(* Logix 5000 project; controller Sucrose_Main Emulate 5570 rev 20.12; software revision 20.01; part 3 of 30 *)
(* tags used below, declared in another part *)
   CIPRemote : Area_Program;
   DATE_TIME : Date_Time;
   Rung_Comment : BOOL;
   SucroseCIP_FILTRATION_ALL_PATHS_Selected : BOOL;
   SucroseCIP_FILTRATION_PATH1_Selected : BOOL;
   SucroseCIP_FILTRATION_PATH2_Selected : BOOL;
   SucroseCIP_FILTRATION_PATH3_Selected : BOOL;
   SucroseCIP_FILTRATION_PATH4_Selected : BOOL;
   SucroseCIP_FILTRATION_REMOTE : CIP_REMOTE;
   SucroseCIP_P230401_REMOTE : CIP_REMOTE;
   SucroseCIP_P230402_REMOTE : CIP_REMOTE;
   SucroseCIP_PAUSED : BOOL;
   SucroseCIP_RECEIVING2_REMOTE : CIP_REMOTE;
   SucroseCIP_RINGMAIN_REMOTE : CIP_REMOTE;
   SucroseCIP_RUNNING : BOOL;
   SucroseCIP_SeatLift_Pulsing : BOOL;
   SucroseFiltration : Area_Program;

        .TMR_LOGIC[5]   // AIR BLOW TIMER
        .CALC_LOGIC[0]   // PRE-FILTER 1 DIFF PRESSURE
        .CALC_LOGIC[1]   // PRE-FILTER 2 DIFF PRESSURE
        .BIT_LOGIC[2].2   // FINAL FILTER 1 SIP STARTED
        .BIT_LOGIC[2].3   // FINAL FILTER 2 SIP STARTED
        .BIT_LOGIC[1].4   // BACKFLUSH ROUTINE ACTIVE
        .BIT_LOGIC[1].5   // AIR BLOW STEP 1 ACTIVE
        .BIT_LOGIC[1].6   // AIR BLOW STEP 2 ACTIVE
        .BIT_LOGIC[1].7   // AIR BLOW STEP 3 ACTIVE
        .BIT_LOGIC[1].8   // INITIAL AIR BLOW COMPLETE
        .BIT_LOGIC[2].0   // PRE FILTER 1 SIP STARTED
        .BIT_LOGIC[0].10   // OK TO START TRANSFER PUMP
        .BIT_LOGIC[1].10   // OK TO START BACKFLUSH PUMP
        .BIT_LOGIC[2].1   // PRE FILTER 2 SIP STARTED
        .BIT_LOGIC[2].5   // SIP STEP ACTIVE
        .BIT_LOGIC[0].5   // PRE FILTER 1 FINAL FILTER 1 PATH ENABLED FOR PRODUCTION
        .BIT_LOGIC[1].17   // AIR BLOW ACTIVE
        .BIT_LOGIC[2].6   // SIP STEP COMPLETE
        .BIT_LOGIC[0].6   // PRE FILTER 1 FINAL FILTER 2 PATH ENABLED FOR PRODUCTION
        .BIT_ALARM[0].11   // FINAL FILTER 1 DIFF PRESSURE ABOVE 40 ALARM
        .BIT_ALARM[0].15   // FINAL FILTER 2 DIFF PRESSURE ABOVE 40 ALARM
        .TMR_ALARM[0]   // PRE FILTER 1 DIFF PRESSURE ABOVE 16 ALARM TIMER
        .BIT_LOGIC[1].0   // PRE FILTER 1 BACKFLUSH STARTED
        .BIT_ALARM[0].0   // PRE FILTER 1 DIFF PRESSURE ABOVE 16 ALARM
        .BIT_ALARM[0].1   // PRE FILTER 1 DIFF PRESSURE ABOVE 20 ALARM
        .BIT_ALARM[0].2   // PRE FILTER 1 DIFF PRESSURE ABOVE 6 ALARM
        .TMR_ALARM[2]   // PRE FILTER 1 DIFF PRESSURE ABOVE 6 ALARM TIMER
        .TMR_ALARM[3]   // PRE FILTER 1 DIFF PRESSURE ABOVE 40 ALARM TIMER
        .BIT_ALARM[0].3   // PRE FILTER 1 DIFF PRESSURE ABOVE 40 ALARM
        .BIT_LOGIC[0].7   // PRE FILTER 2 FINAL FILTER 1 PATH ENABLED FOR PRODUCTION
        .BIT_LOGIC[0].8   // PRE FILTER 2 FINAL FILTER 2 PATH ENABLED FOR PRODUCTION
        .TMR_ALARM[4]   // PRE FILTER 2 DIFF PRESSURE ABOVE 16 ALARM
        .BIT_LOGIC[1].1   // PRE FILTER 2 BACKFLUSH STARTED
        .TMR_ALARM[5]   // PRE FILTER 2 DIFF PRESSURE ABOVE 20 ALARM
        .TMR_ALARM[6]   // PRE FILTER 2 DIFF PRESSURE ABOVE 6 ALARM
        .TMR_ALARM[7]   // PRE FILTER 2 DIFF PRESSURE ABOVE 40 ALARM
        .CALC_LOGIC[2]   // FINAL FILTER 1 DIFF PRESSURE
        .TMR_ALARM[8]   // FINAL FILTER 1 DIFF PRESSURE ABOVE 16 ALARM
        .BIT_LOGIC[1].2   // FINAL FILTER 1 BACKFLUSH STARTED
        .TMR_ALARM[10]   // FINAL FILTER 1 DIFF PRESSURE ABOVE 6 ALARM
        .TMR_ALARM[11]   // FINAL FILTER 1 DIFF PRESSURE ABOVE 40 ALARM
        .CALC_LOGIC[3]   // FINAL FILTER 2 DIFF PRESSURE
        .TMR_ALARM[12]   // FINAL FILTER 2 DIFF PRESSURE ABOVE 16 ALARM
        .BIT_LOGIC[1].3   // FINAL FILTER 2 BACKFLUSH STARTED
        .TMR_ALARM[14]   // FINAL FILTER 2 DIFF PRESSURE ABOVE 6 ALARM
        .BIT_ALARM[0].7   // PRE FILTER 2 DIFF PRESSURE ABOVE 40 ALARM
        .TMR_ALARM[1]   // PRE FILTER 1 DIFF PRESSURE ABOVE 20 ALARM TIMER
        .TMR_ALARM[9]   // FINAL FILTER 1 DIFF PRESSURE ABOVE 20 ALARM
        .TMR_ALARM[13]   // FINAL FILTER 2 DIFF PRESSURE ABOVE 20 ALARM
        .TMR_ALARM[15]   // FINAL FILTER 2 DIFF PRESSURE ABOVE 40 ALARM
        .BIT_LOGIC[0].0   // FILTRATION SKID IN PRODUCTION MODE
        .BIT_LOGIC[0].1   // PRE-FILTER 1 READY FOR PRODUCTION
        .BIT_LOGIC[0].2   // PRE-FILTER 2 READY FOR PRODUCTION
        .BIT_LOGIC[0].3   // FINAL FILTER 1 READY FOR PRODUCTION
        .BIT_LOGIC[0].4   // FINAL FILTER 2 READY FOR PRODUCTION
        .BIT_LOGIC[0].9   // OPEN VENT VALVES ON SELECTED FILTERS
        .BIT_LOGIC[1].9   // BACKFLUSH ROUTINE HOT FLUSH STEP ACTIVE
        .BIT_LOGIC[1].11   // SEND FLUSH TO SCRAP
        .BIT_LOGIC[1].12   // BACKFLUSH DRAIN STEP ACTIVE
        .BIT_LOGIC[1].13   // PRE FILTER 1 CIP BACKFLUSH COMPLETE INTERLOCK TO CIP SKID
        .BIT_LOGIC[1].14   // PRE FILTER 2 CIP BACKFLUSH COMPLETE INTERLOCK TO CIP SKID
        .BIT_LOGIC[1].15   // FINAL FILTER 1 CIP BACKFLUSH COMPLETE INTERLOCK TO CIP SKID
        .BIT_LOGIC[1].16   // FINAL FILTER 2 CIP BACKFLUSH COMPLETE INTERLOCK TO CIP SKID
        .BIT_LOGIC[1].18   // FILTER BACKFLUSH FOR CIP SELECTED
        .BIT_LOGIC[2].4   // STAND ALONE SIP SEQUENCE SELECTED
        .BIT_LOGIC[3].0   // AIR INTEGRITY TEST STARTED FOR FINAL FILTER 1
        .BIT_LOGIC[3].1   // AIR INTEGRITY TEST STARTED FOR FINAL FILTER 2
        .BIT_LOGIC[3].2   // FINAL FILTER INTEGRITY TEST ACTIVE
        .BIT_LOGIC[3].3   // FINAL FILTER INTEGRITY TEST FAILED
        .BIT_LOGIC[3].4   // FINAL FILTER INTEGRITY TEST COMPLETE
        .BIT_LOGIC[3].5   // FINAL FILTER 1 INTEGRITY TEST SELECTED
        .BIT_LOGIC[3].6   // FINAL FILTER 2 INTEGRITY TEST SELECTED
        .TMR_LOGIC[0]   // INITIAL FILTRATION VENTING TIMER
        .TMR_LOGIC[1]   // VENTING AFTER TRANSFER PUMP TIMER
        .TMR_LOGIC[6]   // BACKFLUSH INITIAL FILTRATION VENTING TIMER
        .TMR_LOGIC[7]   // DELAY TO CLOSE VENT VALVE TIMER
        .TMR_LOGIC[8]   // BACKFLUSH SEQUENCE FLUSH ACTIVE TIMER
        .TMR_LOGIC[9]   // BACKFLUSH DRAIN SYSTEM TIMER
        .TMR_LOGIC[10]   // SIP SEQUENCE 250 DEG TIMER
        .TMR_LOGIC[11]   // INITIAL AIR INTEGRITY TEST TIMER
        .TMR_LOGIC[12]   // AIR INTEGRITY TEST ACTIVE TIMER
        .TMR_LOGIC[13]   // SIP SEQUENCE 254 DEG TIMER
        .TMR_LOGIC[14]   // SIP SEQUENCE BELOW TEMP TIMER
        .TMR_LOGIC[15]   // DELAY AFTER CLOSING STEAM VALVE
        .CTR_LOGIC[0]   // PRE FILTER 1 BACKFLUSH COUNTER
        .CTR_LOGIC[1]   // PRE FILTER 2 BACKFLUSH COUNTER
        .CTR_LOGIC[2]   // FINAL FILTER 1 BACKFLUSH COUNTER
        .CTR_LOGIC[3]   // FINAL FILTER 2 BACKFLUSH COUNTER
        .BIT_HMI[0].0   // PRE-FILTER 1 WITH FINAL FILTER 1PATH SELECTED PB
        .BIT_HMI[0].1   // PRE-FILTER 1 WITH FINAL FILTER 2 PATH SELECTED PB
        .BIT_HMI[0].2   // PRE-FILTER 2 WITH FINAL FILTER 1PATH SELECTED PB
        .BIT_HMI[0].3   // PRE-FILTER 2 WITH FINAL FILTER 2 PATH SELECTED PB
        .BIT_HMI[0].4   // FILTER INSTALLED IN PRE FILTER 1 HMI CONFIRMATION
        .BIT_HMI[0].5   // FILTER INSTALLED IN PRE FILTER 2 HMI CONFIRMATION
        .BIT_HMI[0].6   // FILTER INSTALLED IN FINAL FILTER 1 HMI CONFIRMATION
        .BIT_HMI[0].7   // FILTER INSTALLED IN FINAL FILTER 2 HMI CONFIRMATION
        .BIT_HMI[0].8   // PRE FILTER 1 YELLOW FLASHING WARNING ON HMI
        .BIT_HMI[0].9   // PRE FILTER 2 YELLOW FLASHING WARNING ON HMI
        .BIT_HMI[0].10   // FINAL FILTER 1 YELLOW FLASHING WARNING ON HMI
        .BIT_HMI[0].11   // FINAL FILTER 2 YELLOW FLASHING WARNING ON HMI
        .BIT_HMI[0].12   // PRE FILTER 1 RED FLASHING ALARM ON HMI
        .BIT_HMI[0].13   // PRE FILTER 2 RED FLASHING ALARM ON HMI
        .BIT_HMI[0].14   // FIANL FILTER 1 RED FLASHING ALARM ON HMI
        .BIT_HMI[0].15   // FIANL FILTER 2 RED FLASHING ALARM ON HMI
        .BIT_HMI[0].16   // PROMPT FOR PRE FILTER 1 FILTER INSTALLED VISIBILITY
        .BIT_HMI[0].17   // PROMPT FOR PRE FILTER 2 FILTER INSTALLED VISIBILITY
        .BIT_HMI[0].18   // PROMPT FOR FINAL FILTER 1 FILTER INSTALLED VISIBILITY
        .BIT_HMI[0].19   // PROMPT FOR FINAL FILTER 2 FILTER INSTALLED VISIBILITY
        .BIT_HMI[0].20   // PROMPT FOR PRE FILTER 1 FILTER NOT INSTALLED VISIBILITY
        .BIT_HMI[0].21   // PROMPT FOR PRE FILTER 2 FILTER NOT INSTALLED VISIBILITY
        .BIT_HMI[0].22   // PROMPT FOR FINAL FILTER 1 FILTER NOT INSTALLED VISIBILITY
        .BIT_HMI[0].23   // PROMPT FOR FINAL FILTER 2 FILTER NOT INSTALLED VISIBILITY
        .BIT_HMI[0].24   // FILTER SEQUENCE STARTED DISABLE FILTER SELECTION VISABILITY
        .BIT_HMI[0].25   // PROMPT FOR PRE FILTER 1 NEW FILTER INSTALLED VISIBILITY
        .BIT_HMI[0].26   // PROMPT FOR PRE FILTER 2 NEW FILTER INSTALLED VISIBILITY
        .BIT_HMI[0].27   // PROMPT FOR FINAL FILTER 1 NEW FILTER INSTALLED VISIBILITY
        .BIT_HMI[0].28   // PROMPT FOR FINAL FILTER 2 NEW FILTER INSTALLED VISIBILITY
        .BIT_HMI[1].0   // FILTER ROUTINE START PB
        .BIT_HMI[1].1   // BACKFLUSH ROUTINE ABORT PB
        .BIT_HMI[1].2   // FILTER ROUTINE PAUSE PB
        .BIT_HMI[1].5   // PRE FILTER 1 SELECTED FOR BACKFLUSH
        .BIT_HMI[1].6   // PRE FILTER 2 SELECTED FOR BACKFLUSH
        .BIT_HMI[1].7   // FINAL FILTER 1 SELECTED FOR BACKFLUSH
        .BIT_HMI[1].8   // FINAL FILTER 2 SELECTED FOR BACKFLUSH
        .BIT_HMI[1].10   // PRE FILTER 1 SELECTED FOR CIP BACKFLUSH
        .BIT_HMI[1].11   // PRE FILTER 2 SELECTED FOR CIP BACKFLUSH
        .BIT_HMI[1].12   // FINAL FILTER 1 SELECTED FOR CIP BACKFLUSH
        .BIT_HMI[1].13   // FINAL FILTER 2 SELECTED FOR CIP BACKFLUSH
        .BIT_HMI[2].0   // SIP ROUTINE START PB
        .BIT_HMI[2].1   // SIP ROUTINE ABORT PB
        .BIT_HMI[2].5   // PRE FILTER 1 SELECTED FOR SIP
        .BIT_HMI[2].6   // PRE FILTER 2 SELECTED FOR SIP
        .BIT_HMI[2].7   // FINAL FILTER 1 SELECTED FOR SIP
        .BIT_HMI[2].8   // FINAL FILTER 2 SELECTED FOR SIP
        .BIT_HMI[3].0   // AIR INTEGRITY TEST START PB
        .BIT_HMI[3].1   // AIR INTEGRITY TEST ABORT PB
        .BIT_HMI[3].5   // FINAL FILTER 1 SELECTED FOR AIR INTEGRITY TEST
        .BIT_HMI[3].6   // FINAL FILTER 2 SELECTED FOR AIR INTEGRITY TEST
        .STATUS_HMI[1]   // PREFILTER 1 STATUS 0=PROD, 1=AIRBLOW, 2=BACKFLUSH, 3=SIP, 4=INTERG TEST, 5=CIP, 6=SERVICE
        .STATUS_HMI[2]   // PREFILTER 2 STATUS 0=PROD, 1=AIRBLOW, 2=BACKFLUSH, 3=SIP, 4=INTERG TEST, 5=CIP, 6=SERVICE
        .STATUS_HMI[3]   // FINAL FILTER 1 STATUS 0=PROD, 1=AIRBLOW, 2=BACKFLUSH, 3=SIP, 4=INTERG TEST, 5=CIP, 6=SERVICE
        .STATUS_HMI[4]   // FINAL FILTER 2 STATUS 0=PROD, 1=AIRBLOW, 2=BACKFLUSH, 3=SIP, 4=INTERG TEST, 5=CIP, 6=SERVICE
   SucroseReceiving : Area_Program := (TMR_Alarm[0].PRE := 15000, TMR_Alarm[1].PRE := 15000, TMR_Logic[3].PRE := 3000, TMR_Logic[4].PRE := 5000, TMR_Logic[5].PRE := 45000);
        .BIT_LOGIC[0].0   // SUCROSE TANKER QC APPROVED FOR RECEIVING
        .BIT_LOGIC[0].12   // PIG RETURN SEQUENCE ACTIVE
        .BIT_HMI[0].1   // SUCROSE TANKER START TRANSFER PUSHBUTTON PRESSED
        .BIT_HMI[0].2   // STOP TRANSFER REQUEST TO TANKER PUSHBUTTON PRESSED
        .BIT_LOGIC[0].2   // SUCROSE SUPPLY WATER PURGE ENABLED
        .BIT_LOGIC[0].4   // SUCROSE SUPPLY RECEIVING LINE FLUSH COMPLETE BIT
        .BIT_LOGIC[0].5   // SUCROSE SUPPLY RECEIVING LINE WATER PURGE COMPLETE
        .BIT_LOGIC[0].6   // SUCROSE SUPPLY RECEIVING LINE WATER PURGE PREVENT TANK VALVE FROM OPENING
        .BIT_LOGIC[0].7   // PIG LAUNCH SEQUENCE ACTIVE
        .BIT_LOGIC[0].8   // PLACE PIG IN LAUNCH POSITION
        .BIT_LOGIC[0].9   // ACTIVATE V3.1 VALVE TO SET PIG IN POSITION
        .BIT_LOGIC[0].10   // LAUNCH PIG BIT
        .BIT_LOGIC[0].11   // PIG AT RECEIVING STATION
        .BIT_LOGIC[0].13   // PIG BACK IN LAUNCHER. MOVE INTO PRODUCTION POSITION
        .BIT_LOGIC[0].14   // PIG IN PRODUCTION/CIP POSITION BIT
        .TMR_LOGIC[0]   // SUCROSE SUPPLY FLUSH TOTALIZER TIMER
        .TMR_LOGIC[1]   // SUCROSE SUPPLY WATER PURGE TOTALIZER TIMER
        .TMR_LOGIC[2]   // SUCROSE SUPPLY WATER PURGE DELAY SHUTOFF TIMER
        .TMR_LOGIC[3]   // DELAY TO ACTIVATE V3.1 VALVE
        .TMR_LOGIC[4]   // DELAY TO RETURN PIG TO LAUNCHER
        .TMR_LOGIC[5]   // PIPE VENTING TIMER
        .BIT_HMI[0].0   // SUCROSE TANKER QC APPROVED FOR RECEIVING PUSHBUTTON PRESSED
        .BIT_HMI[0].3   // HMI SUCROSE SUPPLY WATER PURGE PUSHBUTTON
        .BIT_HMI[0].4   // LAUNCH PIG HMI PB
        .BIT_HMI[0].5   // START SUCROSE RECEIVING PUMP HMI PB
        .BIT_HMI[1].1   // HMI SUCROSE TANK 1 DISCHARGE ENABLED PUSHBUTTON PRESSED
        .BIT_LOGIC[1].0   // TANK 1 RECEIVING FOR PIG LAUNCH
        .BIT_LOGIC[2].0   // TANK 2 RECEIVING FOR PIG LAUNCH
        .BIT_LOGIC[3].0   // TANK 3 RECEIVING FOR PIG LAUNCH
        .BIT_ALARM[0].0   // RECEIVING LINE NO FLOW, STOP PUMP 1
        .BIT_LOGIC[0].1   // ENABLE SUCROSE RECEIVING PUMP 1
        .BIT_HMI[0].9   // START SUCROSE RECEIVING PUMP 2 HMI PB
        .BIT_LOGIC[0].3   // ENABLE SUCROSE RECEIVING PUMP 2
        .BIT_HMI[0].10   // STOP SUCROSE RECEIVING PUMP 2 HMI PB
        .BIT_HMI[0].8   // USE PLANT PUMP 1 TO RECEIVE SUCROSE SELECTED PB
        .BIT_HMI[0].6   // STOP SUCROSE RECEIVING PUMP 1 HMI PB
        .BIT_HMI[0].11   // USE PLANT PUMP 2 TO RECEIVE SUCROSE SELECTED PB
        .BIT_ALARM[0].1   // RECEIVING LINE NO FLOW, STOP PUMP 2
   SucroseReturn : Area_Program;
   SucroseTanks : Area_Program := (TMR_Alarm[0].PRE := 6000, TMR_Alarm[1].PRE := 3000, TMR_Alarm[2].PRE := 3000, TMR_Alarm[3].PRE := 3000, TMR_Alarm[4].PRE := 30000, TMR_Alarm[5].PRE := 30000, TMR_Alarm[6].PRE := 30000, TMR_Alarm[7].PRE := 30000, TMR_Alarm[8].PRE := 30000, TMR_Alarm[9].PRE := 30000, TMR_Alarm[19].PRE := 5000, TMR_Alarm[20].PRE := 5000, TMR_Alarm[21].PRE := 5000, TMR_Alarm[22].PRE := 5000, TMR_Alarm[23].PRE := 5000, TMR_Alarm[24].PRE := 5000, TMR_Logic[0].PRE := 20000, TMR_Logic[1].PRE := 40000, TMR_Logic[2].PRE := 40000, TMR_Logic[3].PRE := 40000, TMR_Logic[9].PRE := 900000, TMR_Logic[10].PRE := 900000, TMR_Logic[11].PRE := 15000);
        .BIT_LOGIC[3].0   // SUCROSE TANK 3 OK TO RECEIVE TANKER
        .BIT_HMI[2].0   // HMI SUCROSE TANK 2 SELECTED TO RECEIVE TANKER PUSHBUTTON PRESSED
        .BIT_ALARM[0].10   // HTR_76_01_01 HIGH TEMPERATURE ALARM LATCH
        .BIT_LOGIC[1].3   // SUCROSE TANK 1 DISCHARGE ENABLED
        .BIT_LOGIC[1].9   // SUCROSE TANK 1 HEALOUT ENABLED
        .BIT_HMI[3].0   // HMI SUCROSE TANK 3 SELECTED TO RECEIVE TANKER PUSHBUTTON PRESSED
        .BIT_LOGIC[3].1   // SUCROSE TANK 3 TANK IN USE RECEIVING TANKER
        .BIT_LOGIC[1].12   // TANK
        .BIT_LOGIC[3].5   // SUCROSE TANK 3 DISCHARGE ACTIVE
        .BIT_ALARM[0].14   // HTR_76_02_01 LOW TEMPERATURE ALARM LATCH
        .BIT_LOGIC[1].1   // SUCROSE TANK 1 TANK IN USE RECEIVING TANKER
        .BIT_ALARM[0].13   // HTR_76_01_01 LOW TEMPERATURE ALARM LATCH
        .BIT_HMI[1].0   // HMI SUCROSE TANK 1 SELECTED TO RECEIVE TANKER PUSHBUTTON PRESSED
        .BIT_ALARM[0].16   // HTR_76_01_01 LOW FLOW ALARM LATCH
        .BIT_LOGIC[2].2   // SUCROSE TANK 2 READY TO RECEIVE TANKER
        .BIT_LOGIC[1].2   // SUCROSE TANK 1 READY TO RECEIVE TANKER
        .BIT_LOGIC[2].0   // SUCROSE TANK 2 OK TO RECEIVE TANKER
        .BIT_LOGIC[1].5   // SUCROSE TANK 1 DISCHARGE ACTIVE
        .BIT_ALARM[1].3   // TK_23_01_01 SELECTED TANK TOO FULL TO RECEIVE ALARM LATCH
        .BIT_LOGIC[1].0   // SUCROSE TANK 1 OK TO RECEIVE TANKER
        .BIT_LOGIC[3].2   // SUCROSE TANK 3 READY TO RECEIVE TANKER
        .BIT_LOGIC[2].5   // SUCROSE TANK 2 DISCHARGE ACTIVE
        .BIT_LOGIC[2].1   // SUCROSE TANK 2 TANK IN USE RECEIVING TANKER
        .BIT_ALARM[0].11   // HTR_76_02_01 HIGH TEMPERATURE ALARM LATCH
        .BIT_LOGIC[1].4   // TK_23_01_01 READY TO DISCHARGE
        .BIT_ALARM[0].17   // HTR_76_02_01 LOW FLOW ALARM LATCH
        .BIT_ALARM[1].13   // TK_23_02_01 SELECTED TANK TOO FULL TO RECEIVE ALARM LATCH
        .BIT_ALARM[0].12   // HTR_76_03_01 HIGH TEMPERATURE ALARM LATCH
        .BIT_ALARM[0].15   // HTR_76_03_01 LOW TEMPERATURE ALARM LATCH
        .BIT_ALARM[0].18   // HTR_76_03_01 LOW FLOW ALARM LATCH
        .BIT_HMI[1].1   // HMI SUCROSE TANK 1 DISCHARGE ENABLED PUSHBUTTON PRESSED
        .BIT_HMI[2].1   // HMI SUCROSE TANK 2 DISCHARGE ENABLED PUSHBUTTON PRESSED
        .BIT_LOGIC[2].3   // SUCROSE TANK 2 DISCHARGE ENABLED
        .BIT_HMI[3].1   // HMI SUCROSE TANK 3 DISCHARGE ENABLED PUSHBUTTON PRESSED
        .BIT_LOGIC[3].3   // SUCROSE TANK 3 DISCHARGE ENABLED
        .BIT_HMI[1].5   // HMI SUCRSOE TANK 1 HEALOUT ENABLED BIT
        .BIT_LOGIC[2].9   // SUCROSE TANK 2 HEALOUT ENABLED
        .BIT_LOGIC[3].9   // SUCROSE TANK 3 HEALOUT ENABLED
        .BIT_HMI[2].5   // HMI SUCRSOE TANK 2 HEALOUT ENABLED BIT
        .BIT_HMI[3].5   // HMI SUCRSOE TANK 3 HEALOUT ENABLED BIT
        .BIT_LOGIC[2].4   // TK_23_02_01 READY TO DISCHARGE
        .BIT_LOGIC[3].4   // TK_23_03_01 READY TO DISCHARGE
        .BIT_HMI[1].2   // HMI TK_23_01_01 PRIME TO P_23_01_01 PUSHBUTTON PRESSED
        .BIT_LOGIC[2].6   // TK_23_02_01 PRIME ENABLED FOR P_23_01_01 PATH
        .BIT_LOGIC[3].6   // TK_23_03_01 PRIME ENABLED FOR P_23_01_01 PATH
        .BIT_LOGIC[1].6   // TK_23_01_01 PRIME ENABLED FOR P_23_01_01 PATH
        .BIT_HMI[1].3   // HMI TK_23_01_01 PRIME TO P_23_01_02 PUSHBUTTON PRESSED
        .BIT_LOGIC[2].7   // TK_23_02_01 PRIME ENABLED FOR P_23_01_02 PATH
        .BIT_LOGIC[3].7   // TK_23_03_01 PRIME ENABLED FOR P_23_01_02 PATH
        .BIT_LOGIC[1].7   // TK_23_01_01 PRIME ENABLED FOR P_23_01_02 PATH
        .BIT_HMI[2].2   // HMI TK_23_02_01 PRIME TO P_23_01_01 PUSHBUTTON PRESSED
        .BIT_HMI[2].3   // HMI TK_23_02_01 PRIME TO P_23_01_02 PUSHBUTTON PRESSED
        .BIT_HMI[3].2   // HMI TK_23_03_01 PRIME TO P_23_01_01 PUSHBUTTON PRESSED
        .BIT_HMI[3].3   // HMI TK_23_03_01 PRIME TO P_23_01_02 PUSHBUTTON PRESSED
        .BIT_HMI[1].8   // SUCROSE TANK 1 HOLD TANK PB
        .BIT_ALARM[0].0   // NO SUCROSE TANK READY FOR DISCHARGE SUCROSE HEADER WAITING ALARM LATCH
        .BIT_ALARM[0].1   // TK_23_01_01 SELECTED TANK TOO FULL TO RECEIVE ALARM LATCH
        .BIT_ALARM[0].2   // TK_23_02_01 SELECTED TANK TOO FULL TO RECEIVE ALARM LATCH
        .BIT_ALARM[0].3   // TK_23_03_01 SELECTED TANK TOO FULL TO RECEIVE ALARM LATCH
        .BIT_ALARM[0].4   // TK_23_01_01 HIGH TEMPERATURE ALARM LATCH
        .BIT_ALARM[0].5   // TK_23_02_01 HIGH TEMPERATURE ALARM LATCH
        .BIT_ALARM[0].6   // TK_23_03_01 HIGH TEMPERATURE ALARM LATCH
        .BIT_ALARM[0].7   // TK_23_01_01 LOW TEMPERATURE ALARM LATCH
        .BIT_ALARM[0].8   // TK_23_02_01 LOW TEMPERATURE ALARM LATCH
        .BIT_ALARM[0].9   // TK_23_03_01 LOW TEMPERATURE ALARM LATCH
        .BIT_ALARM[1].0   // SUCROSE TANK 1 RUPTURE DISK ALARM
        .BIT_ALARM[1].1   // SUCROSE TANK 2 RUPTURE DISK ALARM
        .BIT_ALARM[1].2   // SUCROSE TANK 3 RUPTURE DISK ALARM
        .BIT_ALARM[1].10   // HTR_76_02_01 HIGH TEMPERATURE ALARM LATCH
        .BIT_ALARM[1].11   // HTR_76_02_01 LOW TEMPERATURE ALARM LATCH
        .BIT_ALARM[1].12   // HTR_76_02_01 LOW FLOW ALARM LATCH
        .BIT_ALARM[1].20   // HTR_76_03_01 HIGH TEMPERATURE ALARM LATCH
        .BIT_ALARM[1].21   // HTR_76_03_01 LOW TEMPERATURE ALARM LATCH
        .BIT_ALARM[1].22   // HTR_76_03_01 LOW FLOW ALARM LATCH
        .BIT_ALARM[1].23   // TK_23_03_01 SELECTED TANK TOO FULL TO RECEIVE ALARM LATCH
        .TMR_ALARM[0]   // NO SUCROSE TANK READY FOR DISCHARGE SUCROSE HEADER WAITING ALARM TIMER
        .TMR_ALARM[1]   // TK_23_01_01 SELECTED TANK TOO FULL TO RECEIVE ALARM TIMER
        .TMR_ALARM[2]   // TK_23_02_01 SELECTED TANK TOO FULL TO RECEIVE ALARM TIMER
        .TMR_ALARM[3]   // TK_23_03_01 SELECTED TANK TOO FULL TO RECEIVE ALARM TIMER
        .TMR_ALARM[4]   // TK_23_01_01 HIGH TEMPERATURE ALARM TIMER
        .TMR_ALARM[5]   // TK_23_02_01 HIGH TEMPERATURE ALARM TIMER
        .TMR_ALARM[6]   // TK_23_03_01 HIGH TEMPERATURE ALARM TIMER
        .TMR_ALARM[7]   // TK_23_01_01 LOW TEMPERATURE ALARM TIMER
        .TMR_ALARM[8]   // TK_23_02_01 LOW TEMPERATURE ALARM TIMER
        .TMR_ALARM[9]   // TK_23_03_01 LOW TEMPERATURE ALARM TIMER
        .TMR_ALARM[10]   // HTR_76_01_01 HIGH TEMPERATURE ALARM TIMER
        .TMR_ALARM[11]   // HTR_76_02_01 HIGH TEMPERATURE ALARM TIMER
        .TMR_ALARM[12]   // HTR_76_03_01 HIGH TEMPERATURE ALARM TIMER
        .TMR_ALARM[13]   // HTR_76_01_01 LOW TEMPERATURE ALARM TIMER
        .TMR_ALARM[14]   // HTR_76_02_01 LOW TEMPERATURE ALARM TIMER
        .TMR_ALARM[15]   // HTR_76_03_01 LOW TEMPERATURE ALARM TIMER
        .TMR_ALARM[16]   // HTR_76_01_01 LOW FLOW ALARM TIMER
        .TMR_ALARM[17]   // HTR_76_02_01 LOW FLOW ALARM TIMER
        .TMR_ALARM[18]   // HTR_76_03_01 LOW FLOW ALARM TIMER
        .BIT_LOGIC[0].0   // SUCROSE TANK SIP SEQUENCE ACTIVE
        .BIT_LOGIC[0].2   // OPEN VENT VALVES ON FILTERS
        .BIT_LOGIC[0].3   // SIP SEQUENCE COMPLETE
        .BIT_LOGIC[0].4   // TANK SIP SEQUENCE ENABLED
        .BIT_LOGIC[1].8   // HMI SUCROSE TANK 1 DRAIN TANK ENABLED
        .BIT_LOGIC[1].10   // TANK 1 SELECTED FOR SIP
        .BIT_LOGIC[1].11   // TANK 1 SIP SEQUENCE ENABLED
        .BIT_LOGIC[2].8   // HMI SUCROSE TANK 2 DRAIN TANK ENABLED
        .BIT_LOGIC[2].10   // TANK 2 SELECTED FOR SIP
        .BIT_LOGIC[2].11   // TANK 2 SIP SEQUENCE ENABLED
        .BIT_LOGIC[3].8   // HMI SUCROSE TANK 3 DRAIN TANK ENABLED
        .BIT_LOGIC[3].10   // TANK 3 SELECTED FOR SIP
        .BIT_LOGIC[3].11   // TANK 3 SIP SEQUENCE ENABLED
        .TMR_LOGIC[0]   // OPEN VENT VALVES ON FILTERS TIMER
        .TMR_LOGIC[1]   // SUCROSE TANK 1 HEALOUT TIMER
        .TMR_LOGIC[2]   // SUCROSE TANK 2 HEALOUT TIMER
        .TMR_LOGIC[3]   // SUCROSE TANK 3 HEALOUT TIMER
        .BIT_HMI[0].0   // SIP SEQUENCE START PB
        .BIT_HMI[0].1   // SIP SEQUENCE ABORT PB
        .BIT_HMI[0].2   // SIP CIRCUIT START PB
        .BIT_HMI[1].4   // HMI SUCROSE TANK 1 DRAIN TANK PUSHBUTTON PRESSED
        .BIT_HMI[1].6   // HMI SUCROSE TANK 1 HEALOUT TIMER RESET PUSHBUTTON
        .BIT_HMI[1].10   // TANK 1 SELECT FOR SIP HMI PB
        .BIT_HMI[2].4   // HMI SUCROSE TANK 2 DRAIN TANK PUSHBUTTON PRESSED
        .BIT_HMI[2].6   // HMI SUCROSE TANK 2 HEALOUT TIMER RESET PUSHBUTTON
        .BIT_HMI[2].10   // TANK 2 SELECT FOR SIP HMI PB
        .BIT_HMI[3].4   // HMI SUCROSE TANK 3 DRAIN TANK PUSHBUTTON PRESSED
        .BIT_HMI[3].6   // HMI SUCROSE TANK 3 HEALOUT TIMER RESET PUSHBUTTON
        .BIT_HMI[3].10   // TANK 3 SELECT FOR SIP HMI PB
        .BIT_HMI[2].8   // SUCROSE TANK 2 HOLD TANK PB
        .BIT_HMI[3].8   // SUCROSE TANK 3 HOLD TANK PB
        .BIT_HMI[2].9   // TRANSFER TO TANK 2 SELECT PB
        .BIT_HMI[3].9   // TRANSFER TO TANK 3 SELECT PB
        .BIT_HMI[1].9   // TRANSFER TO TANK 1 SELECT PB
        .BIT_HMI[1].7   // SUCROSE TANK 1 QC APPROVED PB
        .BIT_HMI[2].7   // SUCROSE TANK 2 QC APPROVED PB
        .BIT_HMI[3].7   // SUCROSE TANK 3 QC APPROVED PB
        .BIT_LOGIC[0].1   // TANK SIP CIRCUIT OK TO SIP
        .BIT_ALARM[0].19   // SUCROSE TANK 1 LOW PRESSURE ALARM
        .BIT_ALARM[0].20   // SUCROSE TANK 2 LOW PRESSURE ALARM
        .BIT_ALARM[0].21   // SUCROSE TANK 3 LOW PRESSURE ALARM
        .BIT_ALARM[0].22   // SUCROSE TANK 1 HIGH PRESSURE ALARM
        .BIT_ALARM[0].23   // SUCROSE TANK 2 HIGH PRESSURE ALARM
        .BIT_ALARM[0].24   // SUCROSE TANK 3 HIGH PRESSURE ALARM TIMER
        .TMR_ALARM[19]   // SUCROSE TANK 1 LOW PRESSURE ALARM TIMER
        .TMR_ALARM[20]   // SUCROSE TANK 2 LOW PRESSURE ALARM TIMER
        .TMR_ALARM[24]   // SUCROSE TANK 3 HIGH PRESSURE ALARM TIMER
        .TMR_ALARM[21]   // SUCROSE TANK 3 LOW PRESSURE ALARM TIMER
        .TMR_ALARM[22]   // SUCROSE TANK 1 HIGH PRESSURE ALARM TIMER
        .TMR_ALARM[23]   // SUCROSE TANK 2 HIGH PRESSURE ALARM TIMER
   SUROSE_HEADER_WATER_PURGE_GALS_PER_SEC : DINT;
   SV130401_AOI : QSI_Discrete_Device := (MM_Enable := 1, Config_Energized_Feedback := 1, Config_Disconnect_Feedback := 1, Config_Energized_Text := 1, Config_MO_ResetOnAlarm := 1, Energize_Permissive := 1, Comment := 1);   // SV-13-04-01 SUCROSE TRANSFER PUMP #1 SEAL WATER FLUSH VALVE
   SV130402_AOI : QSI_Discrete_Device := (MM_Enable := 1, Config_Energized_Feedback := 1, Config_Disconnect_Feedback := 1, Config_Energized_Text := 1, Config_MO_ResetOnAlarm := 1, Energize_Permissive := 1, Comment := 1);   // SV-13-04-02 SUCROSE TRANSFER PUMP #2 SEAL WATER FLUSH VALVE
   SV931101_AOI : QSI_Discrete_Device := (DO_Energize := 1, MM_Enable := 1, Config_MO_ResetOnAlarm := 1, Config_TMR_Alm_Preset_ms := 10000, HMI_Energized := 1, HMI_Disconnect_OK := 1, Energize_Permissive := 1, Energize_Enable := 1, Comment := 1);   // SV-93-11-01 STERILE AIR AUTO VENT FOR FLT-93-11-01 SOLENOID VALVE
   SV931102_AOI : QSI_Discrete_Device := (DO_Energize := 1, MM_Enable := 1, Config_MO_ResetOnAlarm := 1, Config_TMR_Alm_Preset_ms := 10000, HMI_Energized := 1, HMI_Disconnect_OK := 1, Energize_Permissive := 1, Energize_Enable := 1, Comment := 1);   // SV-93-11-02 STERILE AIR AUTO DRAIN FOR FLT-93-11-01 SOLENOID VALVE
   SV931201_AOI : QSI_Discrete_Device := (DO_Energize := 1, MM_Enable := 1, Config_MO_ResetOnAlarm := 1, Config_TMR_Alm_Preset_ms := 10000, HMI_Energized := 1, HMI_Disconnect_OK := 1, Energize_Permissive := 1, Energize_Enable := 1, Comment := 1);   // SV-93-12-01 STERILE AIR AUTO VENT FOR FLT-93-12-01 SOLENOID VALVE
   SV931202_AOI : QSI_Discrete_Device := (DO_Energize := 1, MM_Enable := 1, Config_MO_ResetOnAlarm := 1, Config_TMR_Alm_Preset_ms := 10000, HMI_Energized := 1, HMI_Disconnect_OK := 1, Energize_Permissive := 1, Energize_Enable := 1, Comment := 1);   // SV-93-12-02 STERILE AIR AUTO DRAIN FOR FLT-93-12-02 SOLENOID VALVE
   SV931301_AOI : QSI_Discrete_Device := (DO_Energize := 1, MM_Enable := 1, Config_MO_ResetOnAlarm := 1, Config_TMR_Alm_Preset_ms := 10000, HMI_Energized := 1, HMI_Disconnect_OK := 1, Energize_Permissive := 1, Energize_Enable := 1, Comment := 1);   // SV-93-13-01 STERILE AIR AUTO VENT FOR FLT-93-13-01 SOLENOID VALVE
   SV931302_AOI : QSI_Discrete_Device := (DO_Energize := 1, MM_Enable := 1, Config_MO_ResetOnAlarm := 1, Config_TMR_Alm_Preset_ms := 10000, HMI_Energized := 1, HMI_Disconnect_OK := 1, Energize_Permissive := 1, Energize_Enable := 1, Comment := 1);   // SV-93-13-02 STERILE AIR AUTO DRAIN FOR FLT-93-13-02 SOLENOID VALVE
   TANK1_DATE_TIME : Date_Time;
   TANK2_DATE_TIME : Date_Time;
   TANK3_DATE_TIME : Date_Time;
   temp_toggle : BOOL;
   TK_23_01_01_HEALOUT_TIME_REMAINING : DINT := 40;
   TK_23_01_01_HIGH_LEVEL : DINT := 90;
   TK_23_01_01_HIGH_TEMP : DINT;
   TK_23_01_01_LOW_LEVEL : DINT;
   TK_23_01_01_LOW_TEMP : DINT;
   TK_23_01_01_NO_PRESS_ALARM : BOOL;
   TK_23_01_01_NO_TEMP_ALARM : BOOL := 1;
   TK_23_01_01_RECEIVING_COMPLETE : BOOL;
   TK_23_01_01_TEMP_LEVEL : DINT := 10;
   TK_23_02_01_HEALOUT_TIME_REMAINING : DINT := 40;
   TK_23_02_01_HIGH_LEVEL : DINT;
   TK_23_02_01_HIGH_TEMP : DINT;
   TK_23_02_01_LOW_LEVEL : DINT;
   TK_23_02_01_LOW_TEMP : DINT;
   TK_23_02_01_NO_PRESS_ALARM : BOOL;
   TK_23_02_01_NO_TEMP_ALARM : BOOL := 1;
   TK_23_02_01_RECEIVING_COMPLETE : BOOL;
   TK_23_02_01_TEMP_LEVEL : DINT := 10;
   TK_23_03_01_HEALOUT_TIME_REMAINING : DINT := 40;
   TK_23_03_01_HIGH_LEVEL : DINT;
   TK_23_03_01_HIGH_TEMP : DINT;
   TK_23_03_01_LOW_LEVEL : DINT;
   TK_23_03_01_LOW_TEMP : DINT;
   TK_23_03_01_NO_PRESS_ALARM : BOOL;
   TK_23_03_01_NO_TEMP_ALARM : BOOL := 1;
   TK_23_03_01_RECEIVING_COMPLETE : BOOL;
   TK_23_03_01_TEMP_LEVEL : DINT := 10;
   TMR_SLOW_PLS1 : TIMER := (PRE := 500);
   TMR_SLOW_PLS2 : TIMER := (PRE := 500, ACC := 500);
   toggle : BOOL;
END_VAR

PROGRAM CIP_RemoteArea_AutoLogic   (* main routine MainRoutine *)
VAR
   CIP4_PAUSED : BOOL;
   CIP4_RUNNING : BOOL;
END_VAR

ROUTINE Alarm_Logic   (* ladder *)
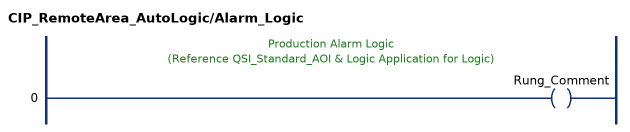
   // Production Alarm Logic
   // (Reference QSI_Standard_AOI & Logic Application for Logic)
   0: OTE(Rung_Comment);
END_ROUTINE

ROUTINE CIP_Filtration_Remote   (* ladder *)
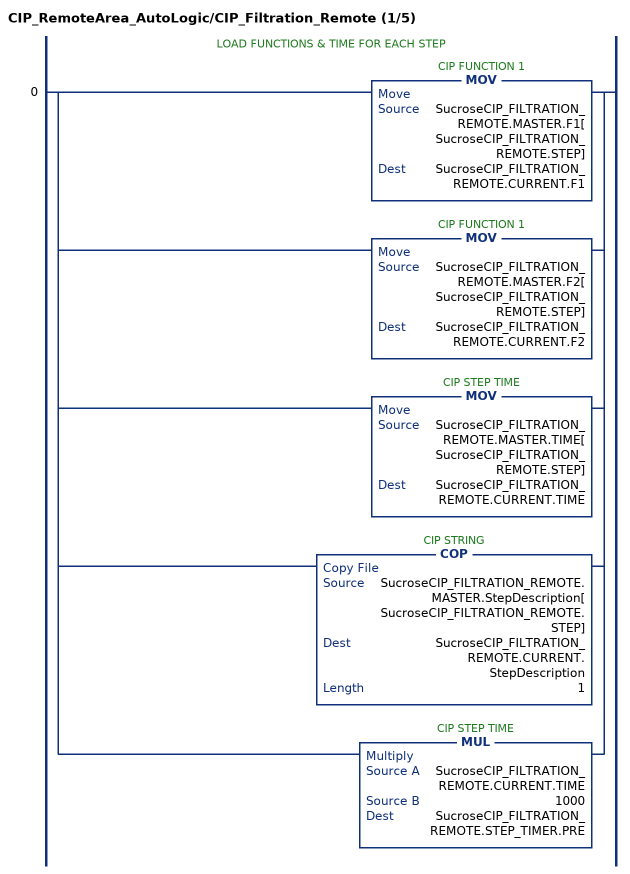
   // LOAD FUNCTIONS & TIME FOR EACH STEP
   0: [MOV(SucroseCIP_FILTRATION_REMOTE.MASTER.F1[SucroseCIP_FILTRATION_REMOTE.STEP],SucroseCIP_FILTRATION_REMOTE.CURRENT.F1) ,MOV(SucroseCIP_FILTRATION_REMOTE.MASTER.F2[SucroseCIP_FILTRATION_REMOTE.STEP],SucroseCIP_FILTRATION_REMOTE.CURRENT.F2) ,MOV(SucroseCIP_FILTRATION_REMOTE.MASTER.TIME[SucroseCIP_FILTRATION_REMOTE.STEP],SucroseCIP_FILTRATION_REMOTE.CURRENT.TIME) ,COP(SucroseCIP_FILTRATION_REMOTE.MASTER.StepDescription[SucroseCIP_FILTRATION_REMOTE.STEP],SucroseCIP_FILTRATION_REMOTE.CURRENT.StepDescription,1) ,MUL(SucroseCIP_FILTRATION_REMOTE.CURRENT.TIME,1000,SucroseCIP_FILTRATION_REMOTE.STEP_TIMER.PRE) ];
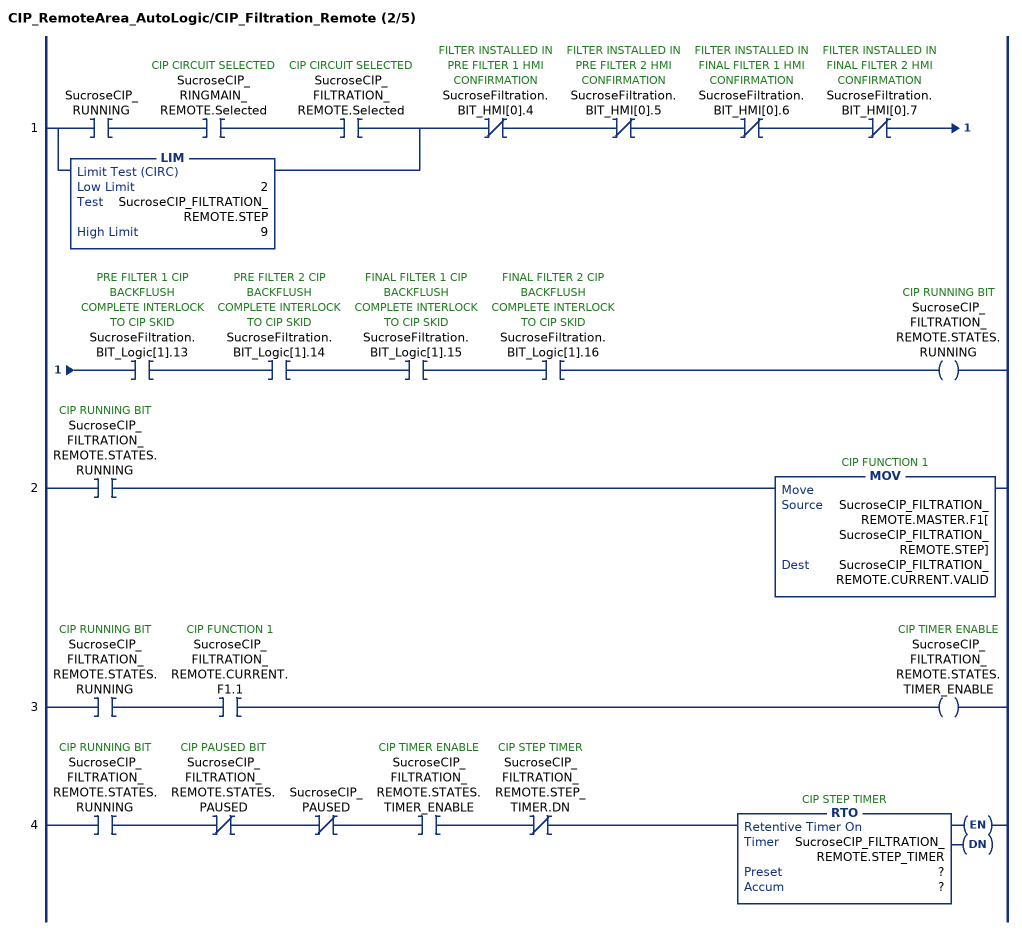
   1: [XIC(SucroseCIP_RUNNING) XIC(SucroseCIP_RINGMAIN_REMOTE.Selected) XIC(SucroseCIP_FILTRATION_REMOTE.Selected) ,LIM(2,SucroseCIP_FILTRATION_REMOTE.STEP,9) ]XIO(SucroseFiltration.BIT_HMI[0].4)XIO(SucroseFiltration.BIT_HMI[0].5)XIO(SucroseFiltration.BIT_HMI[0].6)XIO(SucroseFiltration.BIT_HMI[0].7)XIC(SucroseFiltration.BIT_Logic[1].13)XIC(SucroseFiltration.BIT_Logic[1].14)XIC(SucroseFiltration.BIT_Logic[1].15)XIC(SucroseFiltration.BIT_Logic[1].16)OTE(SucroseCIP_FILTRATION_REMOTE.STATES.RUNNING);
   2: XIC(SucroseCIP_FILTRATION_REMOTE.STATES.RUNNING)MOV(SucroseCIP_FILTRATION_REMOTE.MASTER.F1[SucroseCIP_FILTRATION_REMOTE.STEP],SucroseCIP_FILTRATION_REMOTE.CURRENT.VALID);
   3: XIC(SucroseCIP_FILTRATION_REMOTE.STATES.RUNNING)XIC(SucroseCIP_FILTRATION_REMOTE.CURRENT.F1.1)OTE(SucroseCIP_FILTRATION_REMOTE.STATES.TIMER_ENABLE);
   4: XIC(SucroseCIP_FILTRATION_REMOTE.STATES.RUNNING)XIO(SucroseCIP_FILTRATION_REMOTE.STATES.PAUSED)XIO(SucroseCIP_PAUSED)XIC(SucroseCIP_FILTRATION_REMOTE.STATES.TIMER_ENABLE)XIO(SucroseCIP_FILTRATION_REMOTE.STEP_TIMER.DN)RTO(SucroseCIP_FILTRATION_REMOTE.STEP_TIMER,?,?);
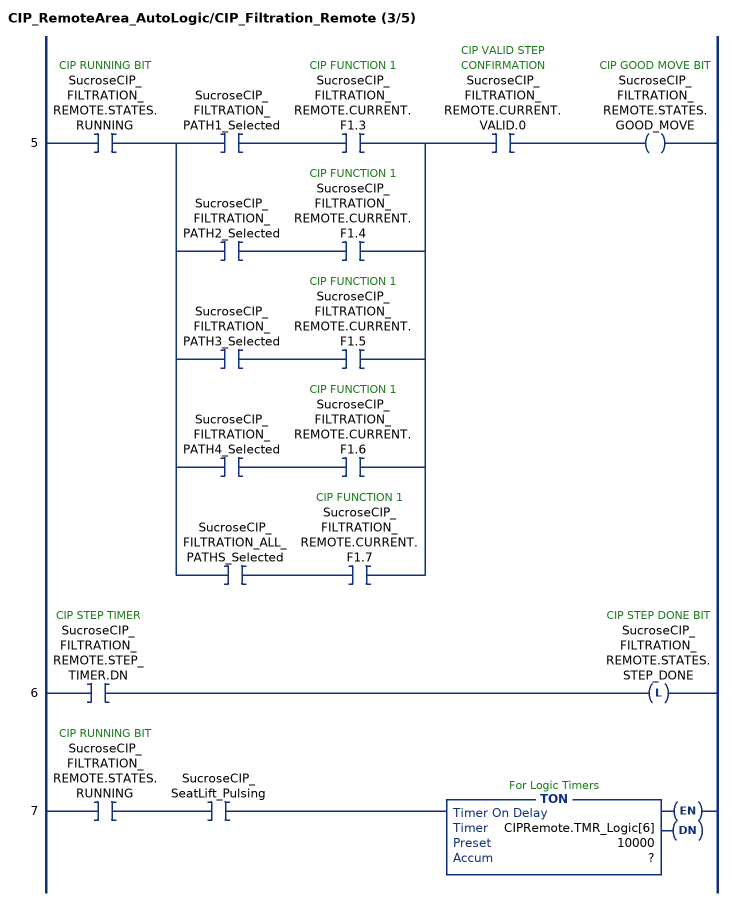
   5: XIC(SucroseCIP_FILTRATION_REMOTE.STATES.RUNNING)[XIC(SucroseCIP_FILTRATION_PATH1_Selected) XIC(SucroseCIP_FILTRATION_REMOTE.CURRENT.F1.3) ,XIC(SucroseCIP_FILTRATION_PATH2_Selected) XIC(SucroseCIP_FILTRATION_REMOTE.CURRENT.F1.4) ,XIC(SucroseCIP_FILTRATION_PATH3_Selected) XIC(SucroseCIP_FILTRATION_REMOTE.CURRENT.F1.5) ,XIC(SucroseCIP_FILTRATION_PATH4_Selected) XIC(SucroseCIP_FILTRATION_REMOTE.CURRENT.F1.6) ,XIC(SucroseCIP_FILTRATION_ALL_PATHS_Selected) XIC(SucroseCIP_FILTRATION_REMOTE.CURRENT.F1.7) ]XIC(SucroseCIP_FILTRATION_REMOTE.CURRENT.VALID.0)OTE(SucroseCIP_FILTRATION_REMOTE.STATES.GOOD_MOVE);
   6: XIC(SucroseCIP_FILTRATION_REMOTE.STEP_TIMER.DN)OTL(SucroseCIP_FILTRATION_REMOTE.STATES.STEP_DONE);
   7: XIC(SucroseCIP_FILTRATION_REMOTE.STATES.RUNNING)XIC(SucroseCIP_SeatLift_Pulsing)TON(CIPRemote.TMR_Logic[6],?,?);
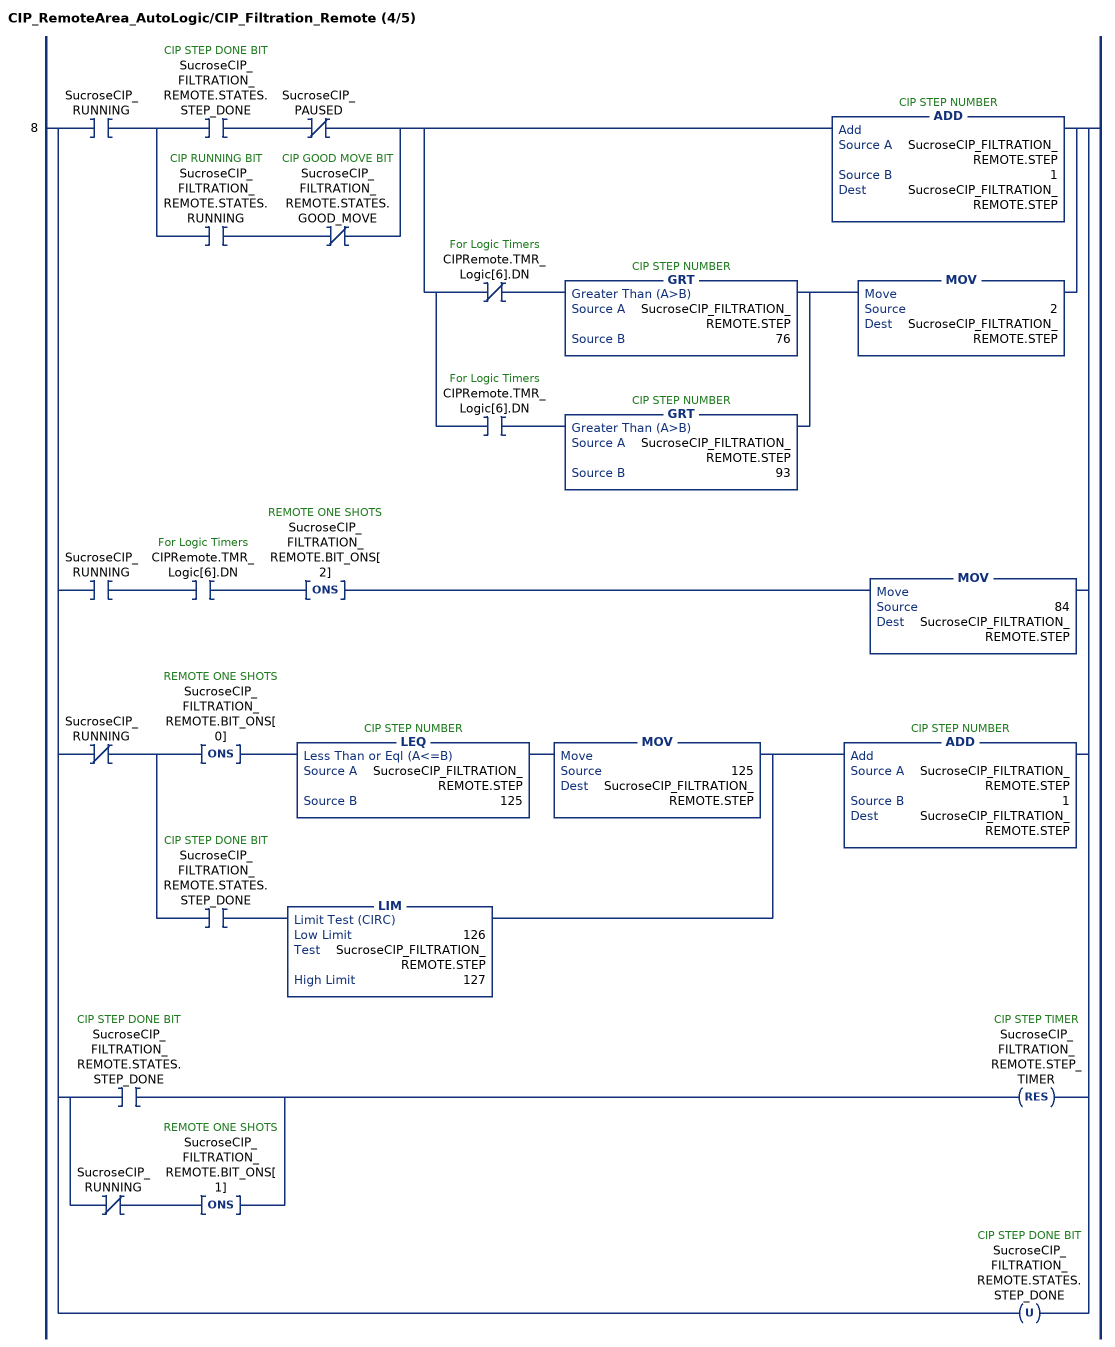
   8: [XIC(SucroseCIP_RUNNING) [XIC(SucroseCIP_FILTRATION_REMOTE.STATES.STEP_DONE) XIO(SucroseCIP_PAUSED) ,XIC(SucroseCIP_FILTRATION_REMOTE.STATES.RUNNING) XIO(SucroseCIP_FILTRATION_REMOTE.STATES.GOOD_MOVE) ] [ADD(SucroseCIP_FILTRATION_REMOTE.STEP,1,SucroseCIP_FILTRATION_REMOTE.STEP) ,[XIO(CIPRemote.TMR_Logic[6].DN) GRT(SucroseCIP_FILTRATION_REMOTE.STEP,76) ,XIC(CIPRemote.TMR_Logic[6].DN) GRT(SucroseCIP_FILTRATION_REMOTE.STEP,93) ] MOV(2,SucroseCIP_FILTRATION_REMOTE.STEP) ] ,XIC(SucroseCIP_RUNNING) XIC(CIPRemote.TMR_Logic[6].DN) ONS(SucroseCIP_FILTRATION_REMOTE.BIT_ONS[2]) MOV(84,SucroseCIP_FILTRATION_REMOTE.STEP) ,XIO(SucroseCIP_RUNNING) [ONS(SucroseCIP_FILTRATION_REMOTE.BIT_ONS[0]) LEQ(SucroseCIP_FILTRATION_REMOTE.STEP,125) MOV(125,SucroseCIP_FILTRATION_REMOTE.STEP) ,XIC(SucroseCIP_FILTRATION_REMOTE.STATES.STEP_DONE) LIM(126,SucroseCIP_FILTRATION_REMOTE.STEP,127) ] ADD(SucroseCIP_FILTRATION_REMOTE.STEP,1,SucroseCIP_FILTRATION_REMOTE.STEP) ,[XIC(SucroseCIP_FILTRATION_REMOTE.STATES.STEP_DONE) ,XIO(SucroseCIP_RUNNING) ONS(SucroseCIP_FILTRATION_REMOTE.BIT_ONS[1]) ] RES(SucroseCIP_FILTRATION_REMOTE.STEP_TIMER) ,OTU(SucroseCIP_FILTRATION_REMOTE.STATES.STEP_DONE) ];
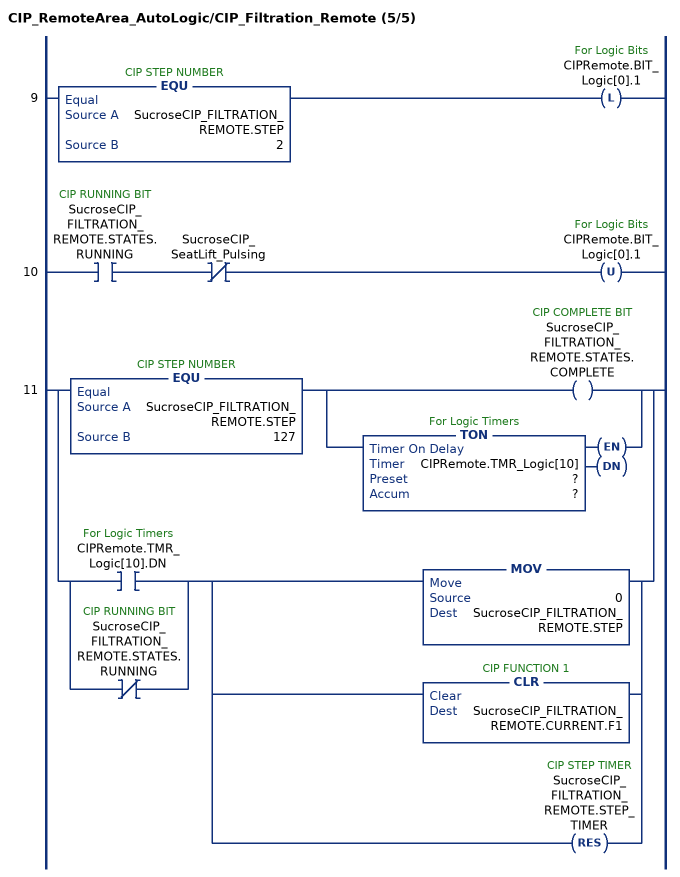
   9: EQU(SucroseCIP_FILTRATION_REMOTE.STEP,2)OTL(CIPRemote.BIT_Logic[0].1);
   10: XIC(SucroseCIP_FILTRATION_REMOTE.STATES.RUNNING)XIO(SucroseCIP_SeatLift_Pulsing)OTU(CIPRemote.BIT_Logic[0].1);
   11: [EQU(SucroseCIP_FILTRATION_REMOTE.STEP,127) [OTE(SucroseCIP_FILTRATION_REMOTE.STATES.COMPLETE) ,TON(CIPRemote.TMR_Logic[10],?,?) ] ,[XIC(CIPRemote.TMR_Logic[10].DN) ,XIO(SucroseCIP_FILTRATION_REMOTE.STATES.RUNNING) ] [MOV(0,SucroseCIP_FILTRATION_REMOTE.STEP) ,CLR(SucroseCIP_FILTRATION_REMOTE.CURRENT.F1) ,RES(SucroseCIP_FILTRATION_REMOTE.STEP_TIMER) ] ];
END_ROUTINE

ROUTINE CIP_P230401_Remote   (* ladder *)
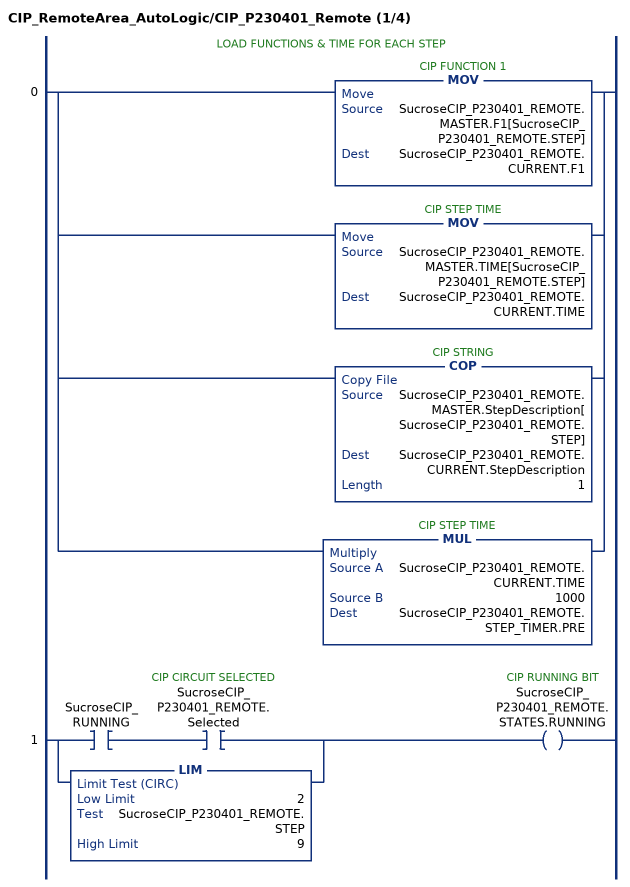
   // LOAD FUNCTIONS & TIME FOR EACH STEP
   0: [MOV(SucroseCIP_P230401_REMOTE.MASTER.F1[SucroseCIP_P230401_REMOTE.STEP],SucroseCIP_P230401_REMOTE.CURRENT.F1) ,MOV(SucroseCIP_P230401_REMOTE.MASTER.TIME[SucroseCIP_P230401_REMOTE.STEP],SucroseCIP_P230401_REMOTE.CURRENT.TIME) ,COP(SucroseCIP_P230401_REMOTE.MASTER.StepDescription[SucroseCIP_P230401_REMOTE.STEP],SucroseCIP_P230401_REMOTE.CURRENT.StepDescription,1) ,MUL(SucroseCIP_P230401_REMOTE.CURRENT.TIME,1000,SucroseCIP_P230401_REMOTE.STEP_TIMER.PRE) ];
   1: [XIC(SucroseCIP_RUNNING) XIC(SucroseCIP_P230401_REMOTE.Selected) ,LIM(2,SucroseCIP_P230401_REMOTE.STEP,9) ]OTE(SucroseCIP_P230401_REMOTE.STATES.RUNNING);
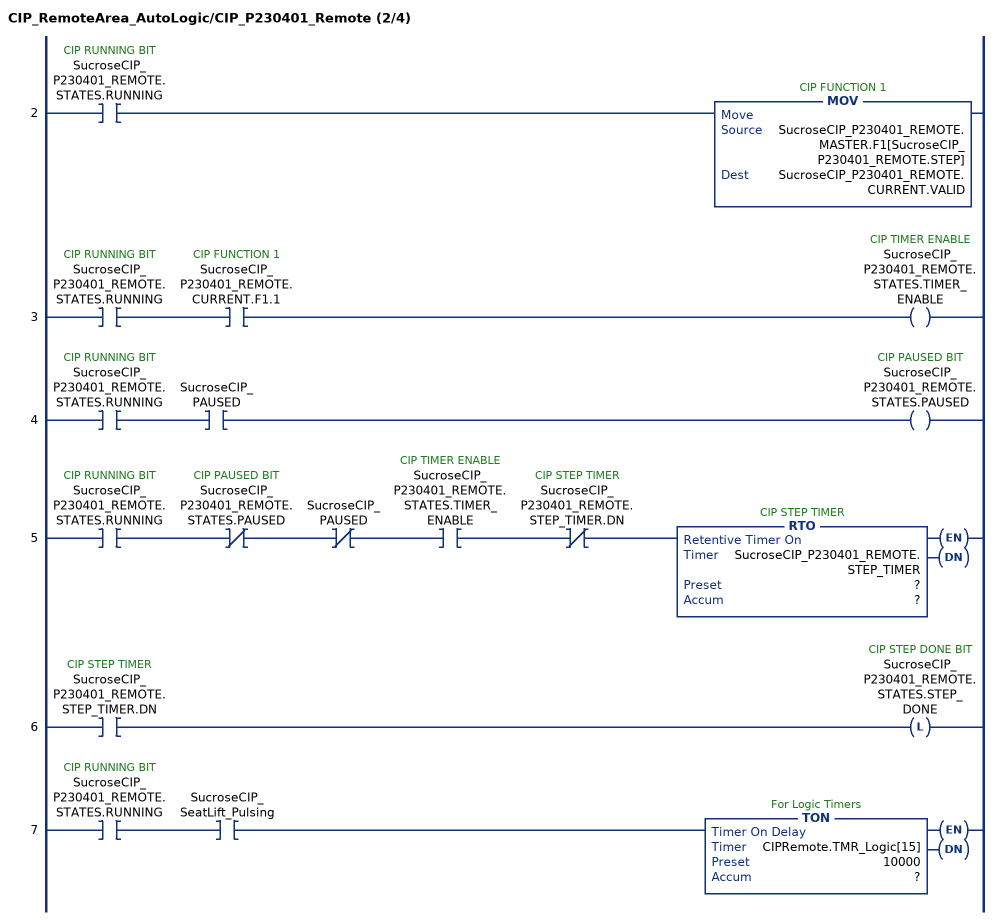
   2: XIC(SucroseCIP_P230401_REMOTE.STATES.RUNNING)MOV(SucroseCIP_P230401_REMOTE.MASTER.F1[SucroseCIP_P230401_REMOTE.STEP],SucroseCIP_P230401_REMOTE.CURRENT.VALID);
   3: XIC(SucroseCIP_P230401_REMOTE.STATES.RUNNING)XIC(SucroseCIP_P230401_REMOTE.CURRENT.F1.1)OTE(SucroseCIP_P230401_REMOTE.STATES.TIMER_ENABLE);
   4: XIC(SucroseCIP_P230401_REMOTE.STATES.RUNNING)XIC(SucroseCIP_PAUSED)OTE(SucroseCIP_P230401_REMOTE.STATES.PAUSED);
   5: XIC(SucroseCIP_P230401_REMOTE.STATES.RUNNING)XIO(SucroseCIP_P230401_REMOTE.STATES.PAUSED)XIO(SucroseCIP_PAUSED)XIC(SucroseCIP_P230401_REMOTE.STATES.TIMER_ENABLE)XIO(SucroseCIP_P230401_REMOTE.STEP_TIMER.DN)RTO(SucroseCIP_P230401_REMOTE.STEP_TIMER,?,?);
   6: XIC(SucroseCIP_P230401_REMOTE.STEP_TIMER.DN)OTL(SucroseCIP_P230401_REMOTE.STATES.STEP_DONE);
   7: XIC(SucroseCIP_P230401_REMOTE.STATES.RUNNING)XIC(SucroseCIP_SeatLift_Pulsing)TON(CIPRemote.TMR_Logic[15],?,?);
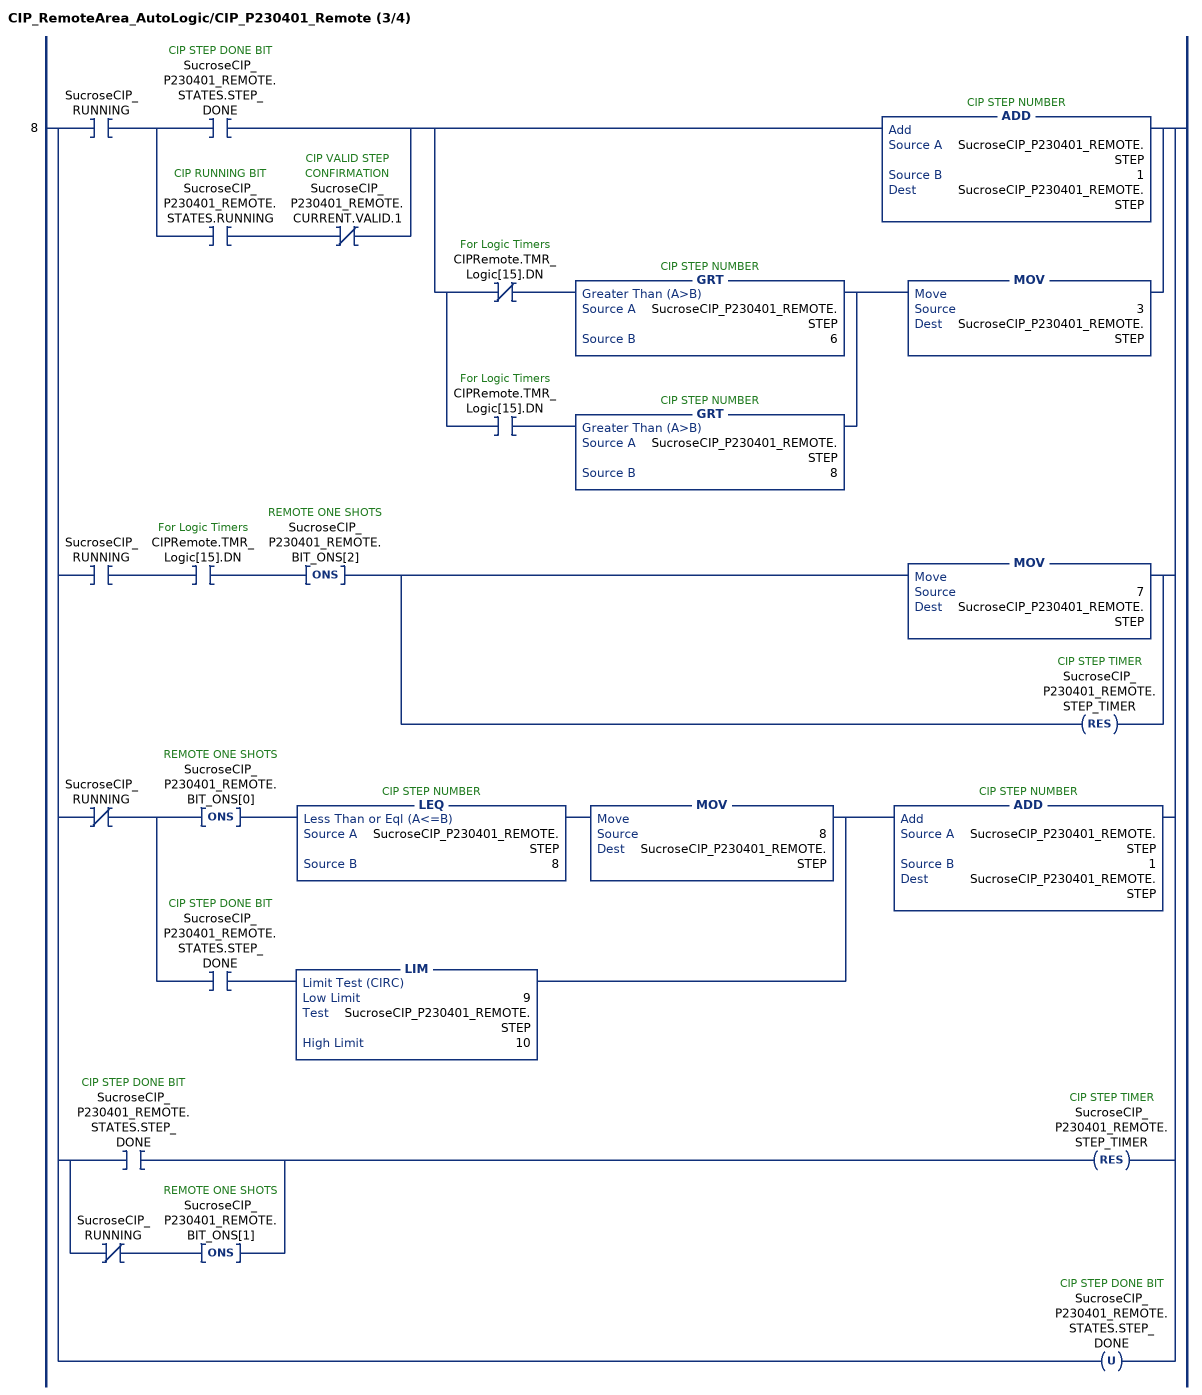
   8: [XIC(SucroseCIP_RUNNING) [XIC(SucroseCIP_P230401_REMOTE.STATES.STEP_DONE) ,XIC(SucroseCIP_P230401_REMOTE.STATES.RUNNING) XIO(SucroseCIP_P230401_REMOTE.CURRENT.VALID.1) ] [ADD(SucroseCIP_P230401_REMOTE.STEP,1,SucroseCIP_P230401_REMOTE.STEP) ,[XIO(CIPRemote.TMR_Logic[15].DN) GRT(SucroseCIP_P230401_REMOTE.STEP,6) ,XIC(CIPRemote.TMR_Logic[15].DN) GRT(SucroseCIP_P230401_REMOTE.STEP,8) ] MOV(3,SucroseCIP_P230401_REMOTE.STEP) ] ,XIC(SucroseCIP_RUNNING) XIC(CIPRemote.TMR_Logic[15].DN) ONS(SucroseCIP_P230401_REMOTE.BIT_ONS[2]) [MOV(7,SucroseCIP_P230401_REMOTE.STEP) ,RES(SucroseCIP_P230401_REMOTE.STEP_TIMER) ] ,XIO(SucroseCIP_RUNNING) [ONS(SucroseCIP_P230401_REMOTE.BIT_ONS[0]) LEQ(SucroseCIP_P230401_REMOTE.STEP,8) MOV(8,SucroseCIP_P230401_REMOTE.STEP) ,XIC(SucroseCIP_P230401_REMOTE.STATES.STEP_DONE) LIM(9,SucroseCIP_P230401_REMOTE.STEP,10) ] ADD(SucroseCIP_P230401_REMOTE.STEP,1,SucroseCIP_P230401_REMOTE.STEP) ,[XIC(SucroseCIP_P230401_REMOTE.STATES.STEP_DONE) ,XIO(SucroseCIP_RUNNING) ONS(SucroseCIP_P230401_REMOTE.BIT_ONS[1]) ] RES(SucroseCIP_P230401_REMOTE.STEP_TIMER) ,OTU(SucroseCIP_P230401_REMOTE.STATES.STEP_DONE) ];
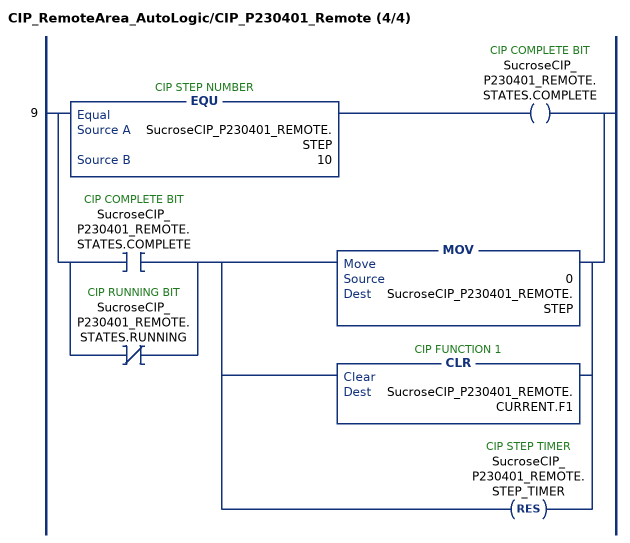
   9: [EQU(SucroseCIP_P230401_REMOTE.STEP,10) OTE(SucroseCIP_P230401_REMOTE.STATES.COMPLETE) ,[XIC(SucroseCIP_P230401_REMOTE.STATES.COMPLETE) ,XIO(SucroseCIP_P230401_REMOTE.STATES.RUNNING) ] [MOV(0,SucroseCIP_P230401_REMOTE.STEP) ,CLR(SucroseCIP_P230401_REMOTE.CURRENT.F1) ,RES(SucroseCIP_P230401_REMOTE.STEP_TIMER) ] ];
END_ROUTINE

ROUTINE CIP_P230402_Remote   (* ladder *)
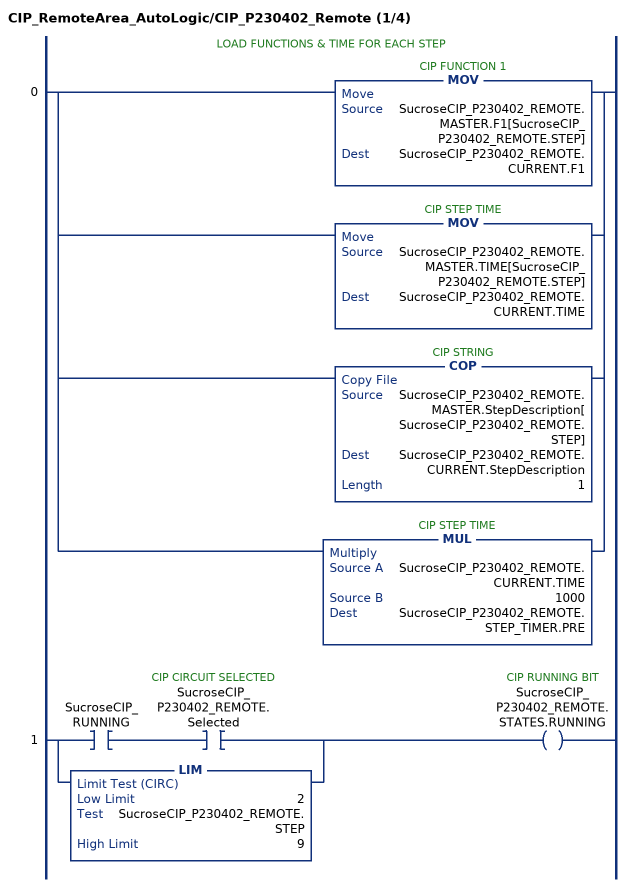
   // LOAD FUNCTIONS & TIME FOR EACH STEP
   0: [MOV(SucroseCIP_P230402_REMOTE.MASTER.F1[SucroseCIP_P230402_REMOTE.STEP],SucroseCIP_P230402_REMOTE.CURRENT.F1) ,MOV(SucroseCIP_P230402_REMOTE.MASTER.TIME[SucroseCIP_P230402_REMOTE.STEP],SucroseCIP_P230402_REMOTE.CURRENT.TIME) ,COP(SucroseCIP_P230402_REMOTE.MASTER.StepDescription[SucroseCIP_P230402_REMOTE.STEP],SucroseCIP_P230402_REMOTE.CURRENT.StepDescription,1) ,MUL(SucroseCIP_P230402_REMOTE.CURRENT.TIME,1000,SucroseCIP_P230402_REMOTE.STEP_TIMER.PRE) ];
   1: [XIC(SucroseCIP_RUNNING) XIC(SucroseCIP_P230402_REMOTE.Selected) ,LIM(2,SucroseCIP_P230402_REMOTE.STEP,9) ]OTE(SucroseCIP_P230402_REMOTE.STATES.RUNNING);
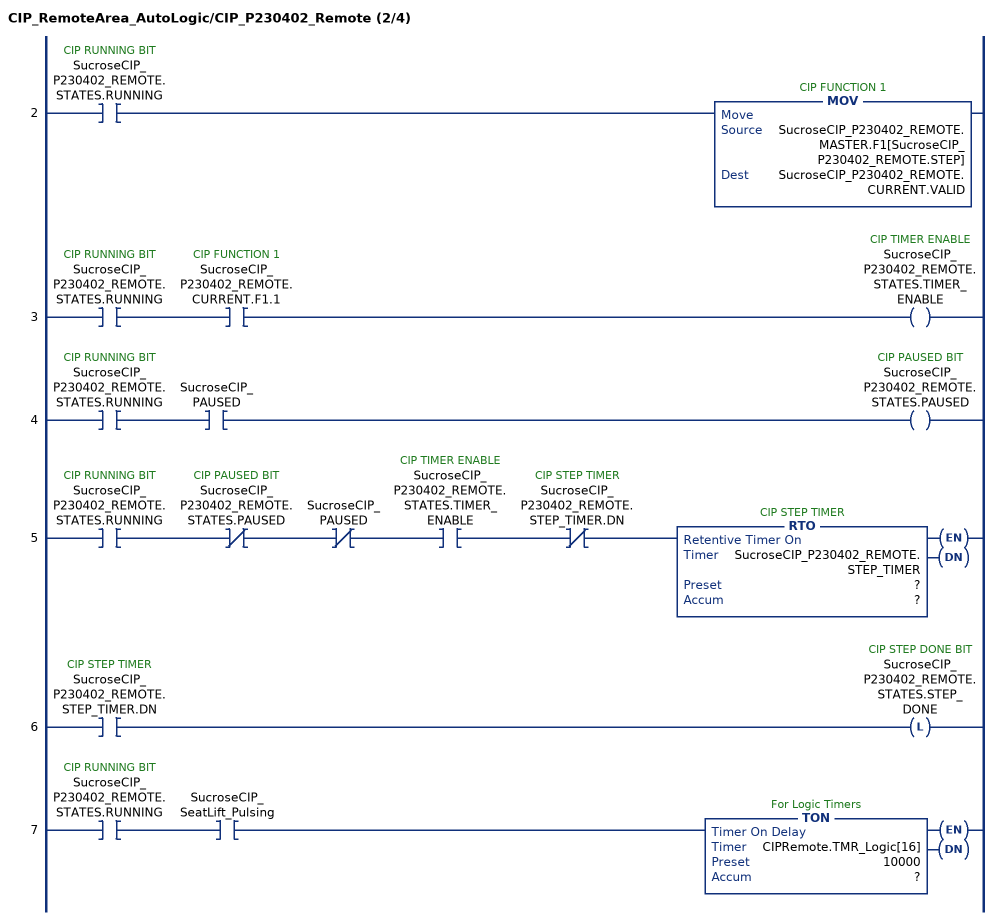
   2: XIC(SucroseCIP_P230402_REMOTE.STATES.RUNNING)MOV(SucroseCIP_P230402_REMOTE.MASTER.F1[SucroseCIP_P230402_REMOTE.STEP],SucroseCIP_P230402_REMOTE.CURRENT.VALID);
   3: XIC(SucroseCIP_P230402_REMOTE.STATES.RUNNING)XIC(SucroseCIP_P230402_REMOTE.CURRENT.F1.1)OTE(SucroseCIP_P230402_REMOTE.STATES.TIMER_ENABLE);
   4: XIC(SucroseCIP_P230402_REMOTE.STATES.RUNNING)XIC(SucroseCIP_PAUSED)OTE(SucroseCIP_P230402_REMOTE.STATES.PAUSED);
   5: XIC(SucroseCIP_P230402_REMOTE.STATES.RUNNING)XIO(SucroseCIP_P230402_REMOTE.STATES.PAUSED)XIO(SucroseCIP_PAUSED)XIC(SucroseCIP_P230402_REMOTE.STATES.TIMER_ENABLE)XIO(SucroseCIP_P230402_REMOTE.STEP_TIMER.DN)RTO(SucroseCIP_P230402_REMOTE.STEP_TIMER,?,?);
   6: XIC(SucroseCIP_P230402_REMOTE.STEP_TIMER.DN)OTL(SucroseCIP_P230402_REMOTE.STATES.STEP_DONE);
   7: XIC(SucroseCIP_P230402_REMOTE.STATES.RUNNING)XIC(SucroseCIP_SeatLift_Pulsing)TON(CIPRemote.TMR_Logic[16],?,?);
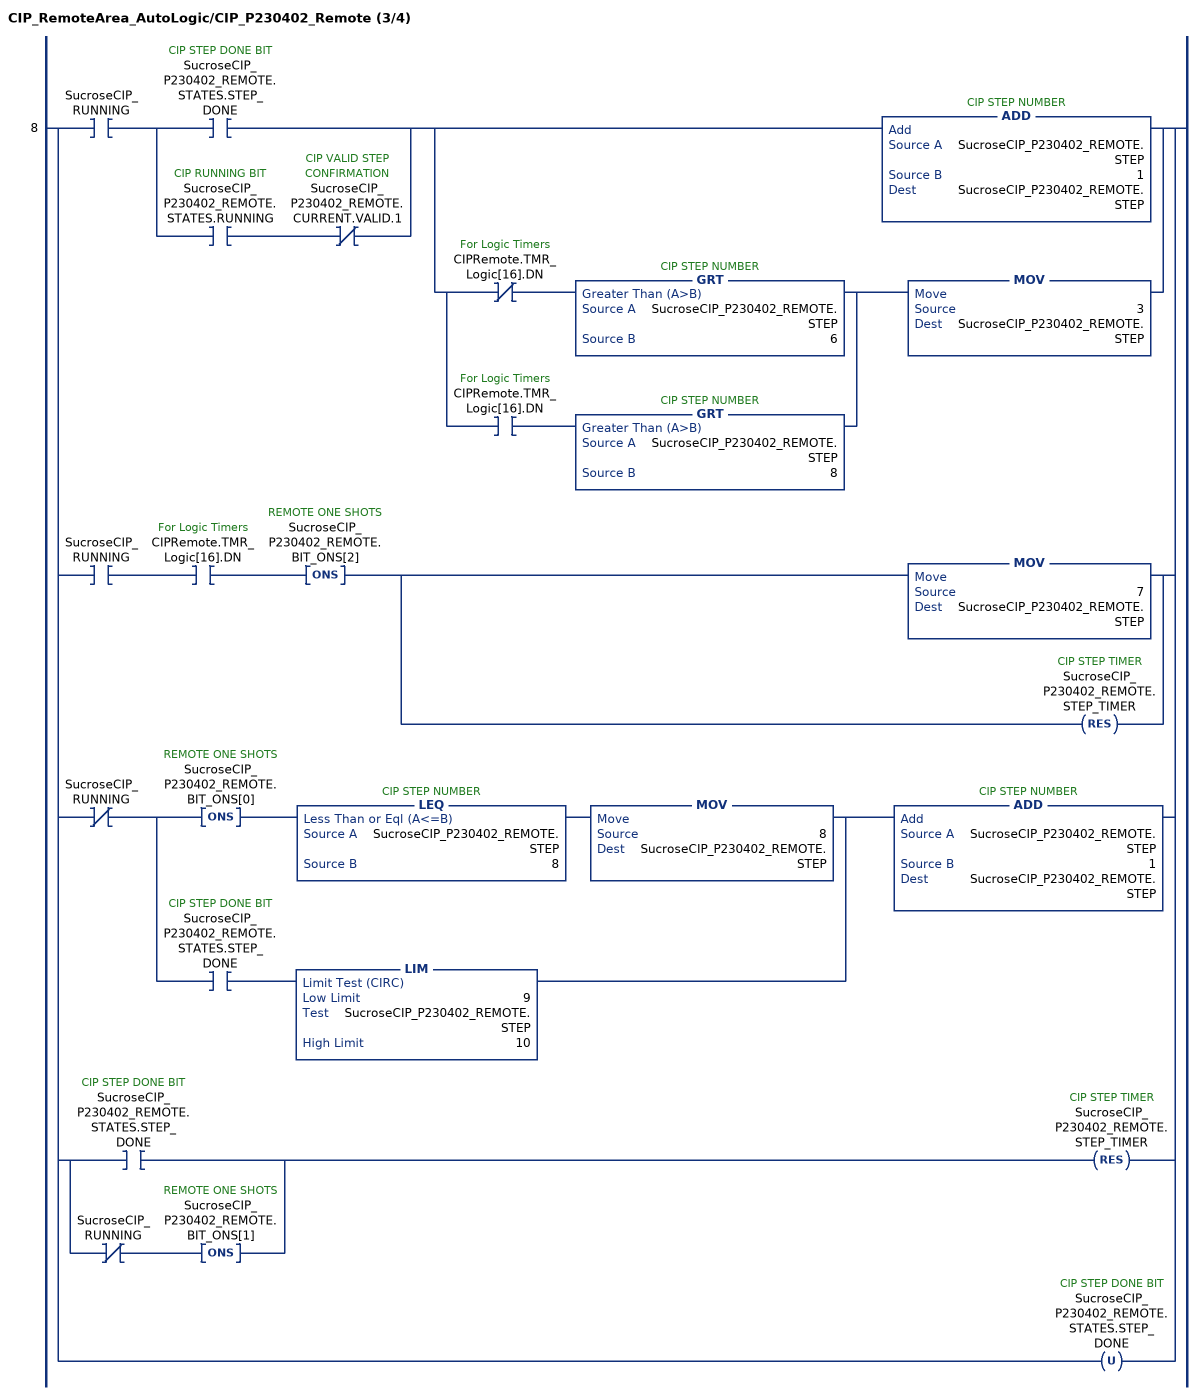
   8: [XIC(SucroseCIP_RUNNING) [XIC(SucroseCIP_P230402_REMOTE.STATES.STEP_DONE) ,XIC(SucroseCIP_P230402_REMOTE.STATES.RUNNING) XIO(SucroseCIP_P230402_REMOTE.CURRENT.VALID.1) ] [ADD(SucroseCIP_P230402_REMOTE.STEP,1,SucroseCIP_P230402_REMOTE.STEP) ,[XIO(CIPRemote.TMR_Logic[16].DN) GRT(SucroseCIP_P230402_REMOTE.STEP,6) ,XIC(CIPRemote.TMR_Logic[16].DN) GRT(SucroseCIP_P230402_REMOTE.STEP,8) ] MOV(3,SucroseCIP_P230402_REMOTE.STEP) ] ,XIC(SucroseCIP_RUNNING) XIC(CIPRemote.TMR_Logic[16].DN) ONS(SucroseCIP_P230402_REMOTE.BIT_ONS[2]) [MOV(7,SucroseCIP_P230402_REMOTE.STEP) ,RES(SucroseCIP_P230402_REMOTE.STEP_TIMER) ] ,XIO(SucroseCIP_RUNNING) [ONS(SucroseCIP_P230402_REMOTE.BIT_ONS[0]) LEQ(SucroseCIP_P230402_REMOTE.STEP,8) MOV(8,SucroseCIP_P230402_REMOTE.STEP) ,XIC(SucroseCIP_P230402_REMOTE.STATES.STEP_DONE) LIM(9,SucroseCIP_P230402_REMOTE.STEP,10) ] ADD(SucroseCIP_P230402_REMOTE.STEP,1,SucroseCIP_P230402_REMOTE.STEP) ,[XIC(SucroseCIP_P230402_REMOTE.STATES.STEP_DONE) ,XIO(SucroseCIP_RUNNING) ONS(SucroseCIP_P230402_REMOTE.BIT_ONS[1]) ] RES(SucroseCIP_P230402_REMOTE.STEP_TIMER) ,OTU(SucroseCIP_P230402_REMOTE.STATES.STEP_DONE) ];
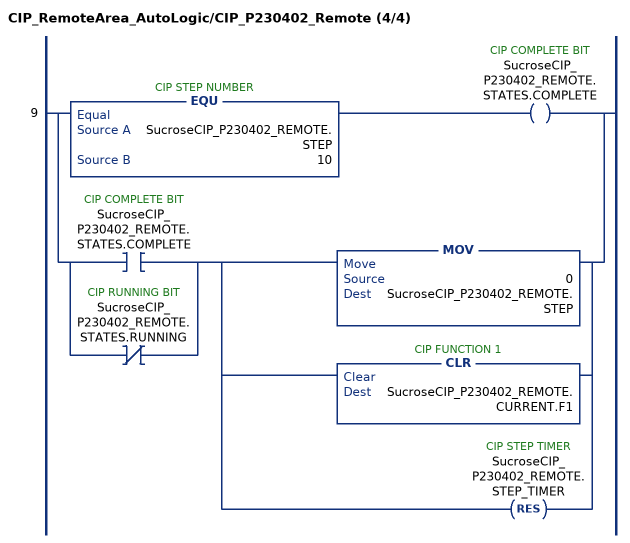
   9: [EQU(SucroseCIP_P230402_REMOTE.STEP,10) OTE(SucroseCIP_P230402_REMOTE.STATES.COMPLETE) ,[XIC(SucroseCIP_P230402_REMOTE.STATES.COMPLETE) ,XIO(SucroseCIP_P230402_REMOTE.STATES.RUNNING) ] [MOV(0,SucroseCIP_P230402_REMOTE.STEP) ,CLR(SucroseCIP_P230402_REMOTE.CURRENT.F1) ,RES(SucroseCIP_P230402_REMOTE.STEP_TIMER) ] ];
END_ROUTINE

ROUTINE CIP_Receiving2_Remote   (* ladder *)
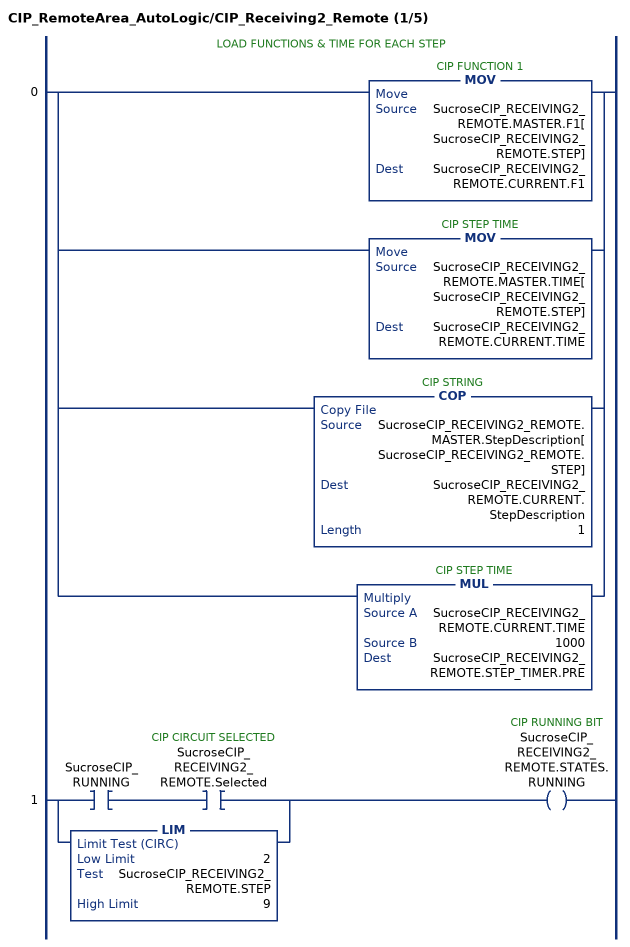
   // LOAD FUNCTIONS & TIME FOR EACH STEP
   0: [MOV(SucroseCIP_RECEIVING2_REMOTE.MASTER.F1[SucroseCIP_RECEIVING2_REMOTE.STEP],SucroseCIP_RECEIVING2_REMOTE.CURRENT.F1) ,MOV(SucroseCIP_RECEIVING2_REMOTE.MASTER.TIME[SucroseCIP_RECEIVING2_REMOTE.STEP],SucroseCIP_RECEIVING2_REMOTE.CURRENT.TIME) ,COP(SucroseCIP_RECEIVING2_REMOTE.MASTER.StepDescription[SucroseCIP_RECEIVING2_REMOTE.STEP],SucroseCIP_RECEIVING2_REMOTE.CURRENT.StepDescription,1) ,MUL(SucroseCIP_RECEIVING2_REMOTE.CURRENT.TIME,1000,SucroseCIP_RECEIVING2_REMOTE.STEP_TIMER.PRE) ];
   1: [XIC(SucroseCIP_RUNNING) XIC(SucroseCIP_RECEIVING2_REMOTE.Selected) ,LIM(2,SucroseCIP_RECEIVING2_REMOTE.STEP,9) ]OTE(SucroseCIP_RECEIVING2_REMOTE.STATES.RUNNING);
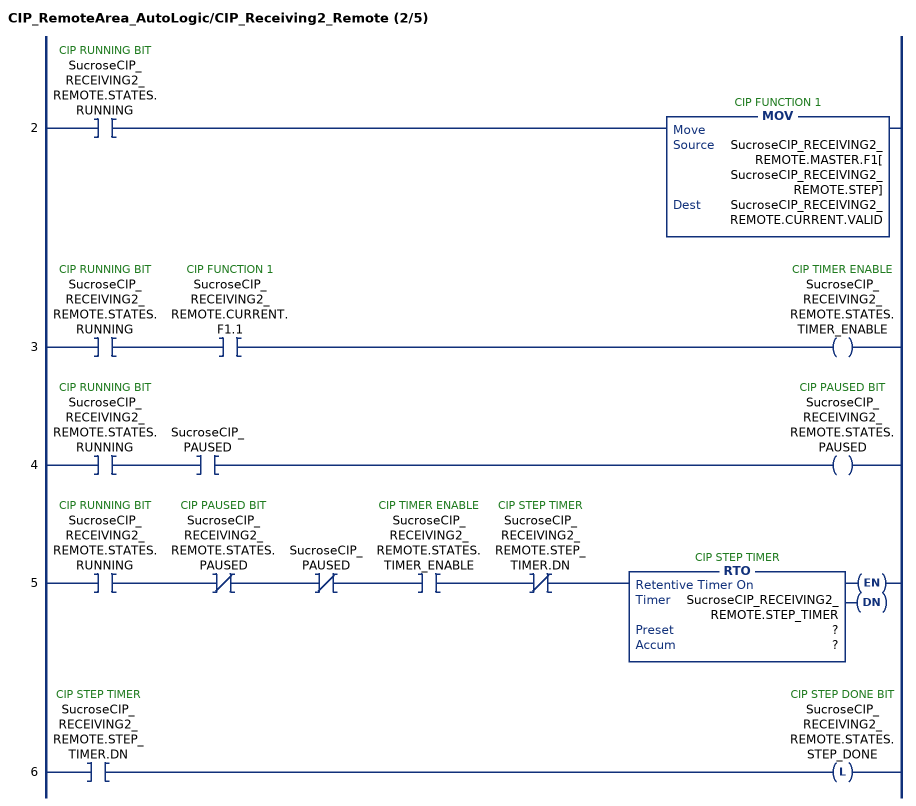
   2: XIC(SucroseCIP_RECEIVING2_REMOTE.STATES.RUNNING)MOV(SucroseCIP_RECEIVING2_REMOTE.MASTER.F1[SucroseCIP_RECEIVING2_REMOTE.STEP],SucroseCIP_RECEIVING2_REMOTE.CURRENT.VALID);
   3: XIC(SucroseCIP_RECEIVING2_REMOTE.STATES.RUNNING)XIC(SucroseCIP_RECEIVING2_REMOTE.CURRENT.F1.1)OTE(SucroseCIP_RECEIVING2_REMOTE.STATES.TIMER_ENABLE);
   4: XIC(SucroseCIP_RECEIVING2_REMOTE.STATES.RUNNING)XIC(SucroseCIP_PAUSED)OTE(SucroseCIP_RECEIVING2_REMOTE.STATES.PAUSED);
   5: XIC(SucroseCIP_RECEIVING2_REMOTE.STATES.RUNNING)XIO(SucroseCIP_RECEIVING2_REMOTE.STATES.PAUSED)XIO(SucroseCIP_PAUSED)XIC(SucroseCIP_RECEIVING2_REMOTE.STATES.TIMER_ENABLE)XIO(SucroseCIP_RECEIVING2_REMOTE.STEP_TIMER.DN)RTO(SucroseCIP_RECEIVING2_REMOTE.STEP_TIMER,?,?);
   6: XIC(SucroseCIP_RECEIVING2_REMOTE.STEP_TIMER.DN)OTL(SucroseCIP_RECEIVING2_REMOTE.STATES.STEP_DONE);
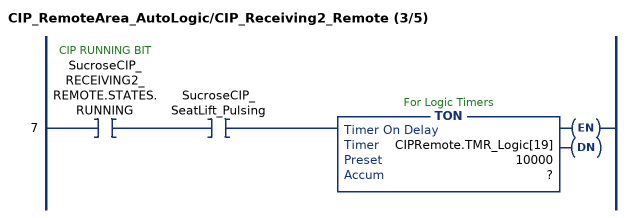
   7: XIC(SucroseCIP_RECEIVING2_REMOTE.STATES.RUNNING)XIC(SucroseCIP_SeatLift_Pulsing)TON(CIPRemote.TMR_Logic[19],?,?);
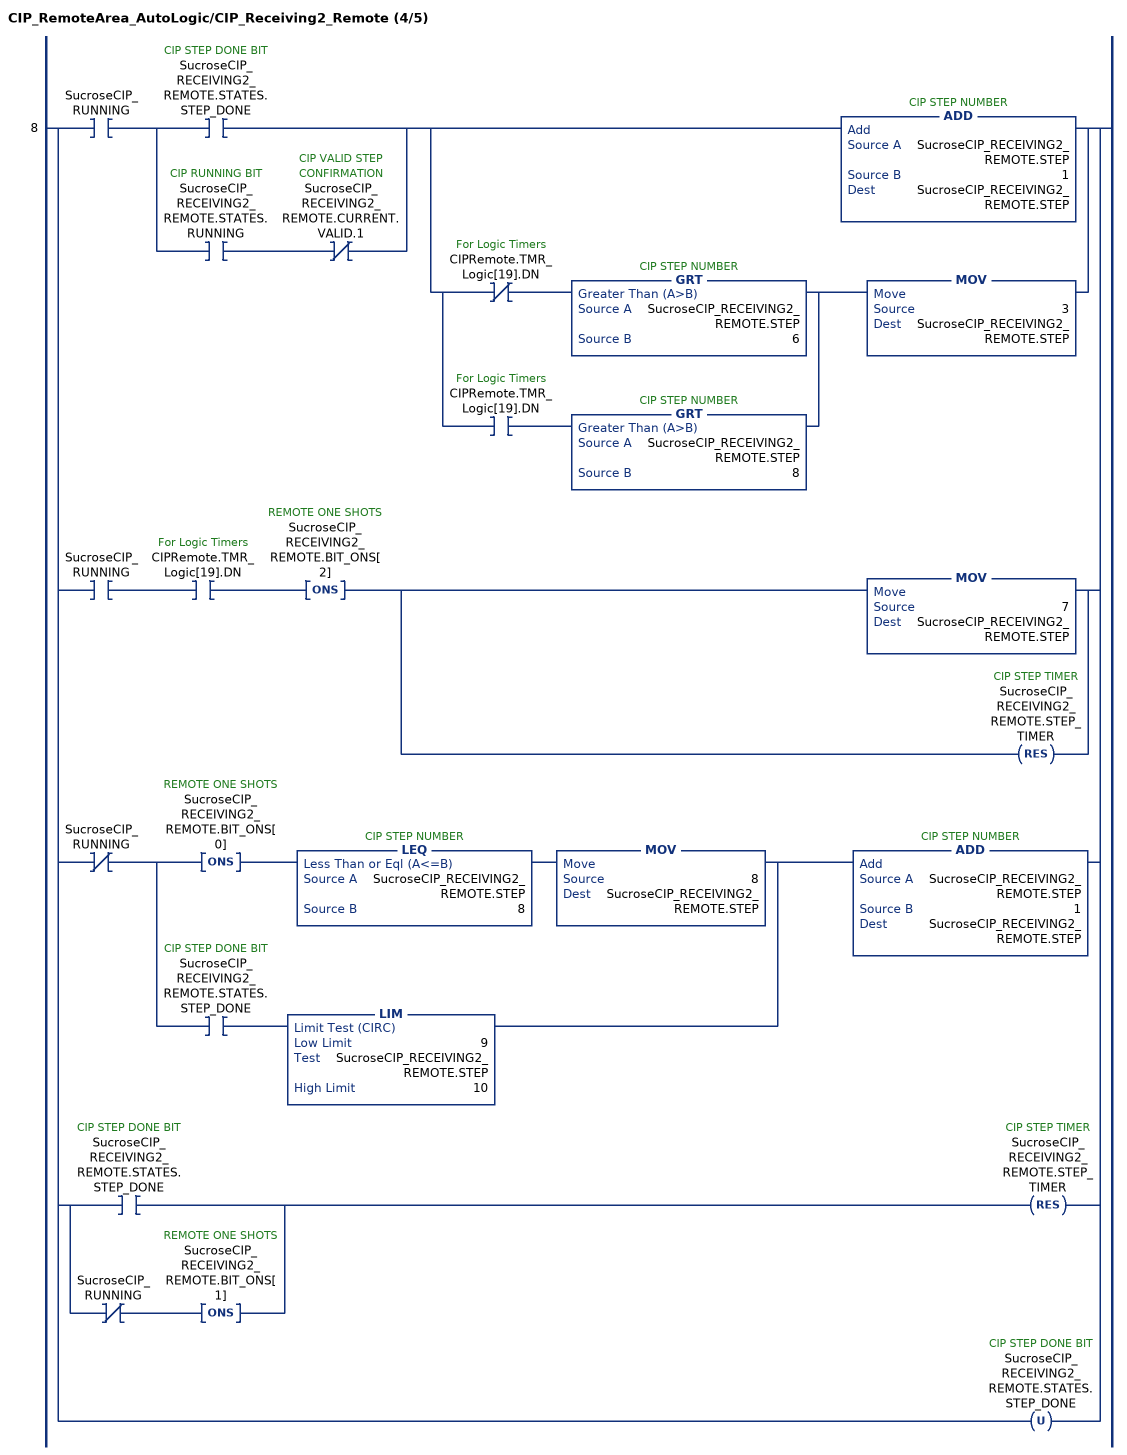
   8: [XIC(SucroseCIP_RUNNING) [XIC(SucroseCIP_RECEIVING2_REMOTE.STATES.STEP_DONE) ,XIC(SucroseCIP_RECEIVING2_REMOTE.STATES.RUNNING) XIO(SucroseCIP_RECEIVING2_REMOTE.CURRENT.VALID.1) ] [ADD(SucroseCIP_RECEIVING2_REMOTE.STEP,1,SucroseCIP_RECEIVING2_REMOTE.STEP) ,[XIO(CIPRemote.TMR_Logic[19].DN) GRT(SucroseCIP_RECEIVING2_REMOTE.STEP,6) ,XIC(CIPRemote.TMR_Logic[19].DN) GRT(SucroseCIP_RECEIVING2_REMOTE.STEP,8) ] MOV(3,SucroseCIP_RECEIVING2_REMOTE.STEP) ] ,XIC(SucroseCIP_RUNNING) XIC(CIPRemote.TMR_Logic[19].DN) ONS(SucroseCIP_RECEIVING2_REMOTE.BIT_ONS[2]) [MOV(7,SucroseCIP_RECEIVING2_REMOTE.STEP) ,RES(SucroseCIP_RECEIVING2_REMOTE.STEP_TIMER) ] ,XIO(SucroseCIP_RUNNING) [ONS(SucroseCIP_RECEIVING2_REMOTE.BIT_ONS[0]) LEQ(SucroseCIP_RECEIVING2_REMOTE.STEP,8) MOV(8,SucroseCIP_RECEIVING2_REMOTE.STEP) ,XIC(SucroseCIP_RECEIVING2_REMOTE.STATES.STEP_DONE) LIM(9,SucroseCIP_RECEIVING2_REMOTE.STEP,10) ] ADD(SucroseCIP_RECEIVING2_REMOTE.STEP,1,SucroseCIP_RECEIVING2_REMOTE.STEP) ,[XIC(SucroseCIP_RECEIVING2_REMOTE.STATES.STEP_DONE) ,XIO(SucroseCIP_RUNNING) ONS(SucroseCIP_RECEIVING2_REMOTE.BIT_ONS[1]) ] RES(SucroseCIP_RECEIVING2_REMOTE.STEP_TIMER) ,OTU(SucroseCIP_RECEIVING2_REMOTE.STATES.STEP_DONE) ];
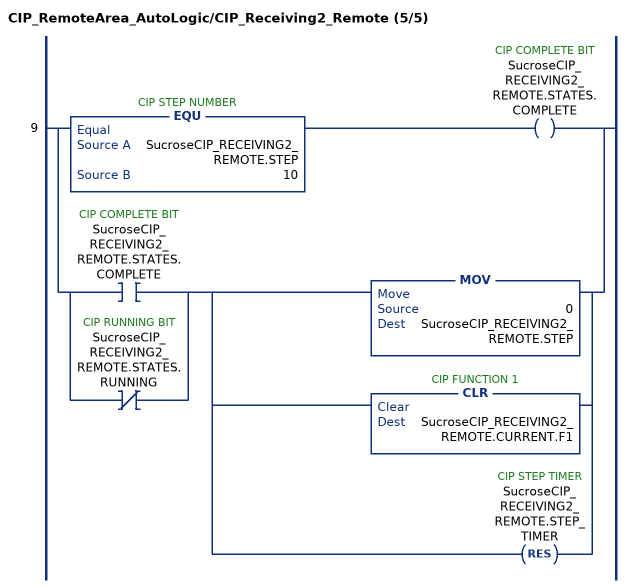
   9: [EQU(SucroseCIP_RECEIVING2_REMOTE.STEP,10) OTE(SucroseCIP_RECEIVING2_REMOTE.STATES.COMPLETE) ,[XIC(SucroseCIP_RECEIVING2_REMOTE.STATES.COMPLETE) ,XIO(SucroseCIP_RECEIVING2_REMOTE.STATES.RUNNING) ] [MOV(0,SucroseCIP_RECEIVING2_REMOTE.STEP) ,CLR(SucroseCIP_RECEIVING2_REMOTE.CURRENT.F1) ,RES(SucroseCIP_RECEIVING2_REMOTE.STEP_TIMER) ] ];
END_ROUTINE
